LIN {X 0,Y 227.48,Z 413.452,A -85,B 0,C 180,E1 -20071.549,E2 -20071.549} C_VEL
LIN {X 0,Y 229.431,Z 419.011,A -85,B 0,C 180,E1 -20072.113,E2 -20072.113} C_VEL
LIN {X 0,Y 232.669,Z 428.465,A -85,B 0,C 180,E1 -20073.214,E2 -20073.214} C_VEL
LIN {X 0,Y 235.611,Z 440.17,A -85,B 0,C 180,E1 -20074.705,E2 -20074.705} C_VEL
LIN {X 0,Y 237.998,Z 451.953,A -85,B 0,C 180,E1 -20076.482,E2 -20076.482} C_VEL
LIN {X 0,Y 238.523,Z 456.323,A -85,B 0,C 180,E1 -20077.194,E2 -20077.194} C_VEL
LIN {X 0,Y 236.555,Z 467.31,A -85,B 0,C 180,E1 -20078.946,E2 -20078.946} C_VEL
LIN {X 0,Y 234.438,Z 477.678,A -85,B 0,C 180,E1 -20081.018,E2 -20081.018} C_VEL
LIN {X 0,Y 232.639,Z 485.999,A -85,B 0,C 180,E1 -20083.096,E2 -20083.096} C_VEL
LIN {X 0,Y 230.834,Z 493.681,A -85,B 0,C 180,E1 -20085.45,E2 -20085.45} C_VEL
LIN {X 0,Y 229.18,Z 500.557,A -85,B 0,C 180,E1 -20088.076,E2 -20088.076} C_VEL
LIN {X 0,Y 227.975,Z 506.106,A -85,B 0,C 180,E1 -20090.764,E2 -20090.764} C_VEL
LIN {X 0,Y 226.971,Z 510.814,A -85,B 0,C 180,E1 -20093.737,E2 -20093.737} C_VEL
LIN {X 0,Y 226.477,Z 513.304,A -85,B 0,C 180,E1 -20095.851,E2 -20095.851} C_VEL
LIN {X 0,Y 226.081,Z 515.094,A -85,B 0,C 180,E1 -20097.794,E2 -20097.794} C_VEL
LIN {X 0,Y 225.853,Z 516.41,A -85,B 0,C 180,E1 -20099.86,E2 -20099.86} C_VEL
LIN {X 0,Y 225.805,Z 517.379,A -85,B 0,C 180,E1 -20102.822,E2 -20102.822} C_VEL
LIN {X 0,Y 226.172,Z 517.171,A -85,B 0,C 180,E1 -20106.185,E2 -20106.185} C_VEL
LIN {X 0,Y 226.927,Z 515.743,A -85,B 0,C 180,E1 -20109.262,E2 -20109.262} C_VEL
LIN {X 0,Y 228.213,Z 512.694,A -85,B 0,C 180,E1 -20112.649,E2 -20112.649} C_VEL
LIN {X 0,Y 229.437,Z 509.335,A -85,B 0,C 180,E1 -20115.208,E2 -20115.208} C_VEL
LIN {X 0,Y 231.319,Z 504.308,A -85,B 0,C 180,E1 -20118.055,E2 -20118.055} C_VEL
LIN {X 0,Y 233.64,Z 497.907,A -85,B 0,C 180,E1 -20120.825,E2 -20120.825} C_VEL
LIN {X 0,Y 236.35,Z 489.874,A -85,B 0,C 180,E1 -20123.508,E2 -20123.508} C_VEL
LIN {X 0,Y 239.203,Z 480.611,A -85,B 0,C 180,E1 -20125.926,E2 -20125.926} C_VEL
LIN {X 0,Y 241.778,Z 471.395,A -85,B 0,C 180,E1 -20127.84,E2 -20127.84} C_VEL
LIN {X 0,Y 243.706,Z 463.116,A -85,B 0,C 180,E1 -20129.259,E2 -20129.259} C_VEL
LIN {X 0,Y 242.372,Z 453.565,A -85,B 0,C 180,E1 -20131.179,E2 -20131.179} C_VEL
LIN {X 0,Y 240.028,Z 444.017,A -85,B 0,C 180,E1 -20133.009,E2 -20133.009} C_VEL
LIN {X 0,Y 237.284,Z 435.697,A -85,B 0,C 180,E1 -20134.566,E2 -20134.566} C_VEL
LIN {X 0,Y 232.657,Z 425.144,A -85,B 0,C 180,E1 -20136.583,E2 -20136.583} C_VEL
LIN {X 0,Y 230.235,Z 420.752,A -85,B 0,C 180,E1 -20137.483,E2 -20137.483} C_VEL
LIN {X 0,Y 228.674,Z 417.665,A -85,B 0,C 180,E1 -20138.078,E2 -20138.078} C_VEL
LIN {X 0,Y 228.509,Z 416.855,A -85,B 0,C 180,E1 -20138.248,E2 -20138.248} C_VEL
LIN {X 0,Y 228.454,Z 415.047,A -85,B 0,C 180,E1 -20142.487,E2 -20142.487} C_VEL
LIN {X 0,Y 228.344,Z 413.795,A -85,B 0,C 180,E1 -20145.745,E2 -20145.745} C_VEL
LIN {X 0,Y 228.264,Z 412.058,A -85,B 0,C 180,E1 -20151.144,E2 -20151.144} C_VEL
LIN {X 0,Y 228.322,Z 412.042,A -85,B 0,C 180,E1 -20152.927,E2 -20152.927} C_VEL
LIN {X 0,Y 228.552,Z 412.016,A -85,B 0,C 180,E1 -20158.238,E2 -20158.238} C_VEL
LIN {X 0,Y 228.552,Z 412.013,A -85,B 0,C 180,E1 -20161.762,E2 -20161.762} C_VEL
LIN {X 0,Y 228.321,Z 412.042,A -85,B 0,C 180,E1 -20167.072,E2 -20167.072} C_VEL
LIN {X 0,Y 228.143,Z 412.061,A -85,B 0,C 180,E1 -20170.651,E2 -20170.651} C_VEL
LIN {X 0,Y 228.06,Z 412.073,A -85,B 0,C 180,E1 -20174.272,E2 -20174.272} C_VEL
LIN {X 0,Y 228.001,Z 412.082,A -85,B 0,C 180,E1 -20177.953,E2 -20177.953} C_VEL
LIN {X 0,Y 227.994,Z 412.377,A -85,B 0,C 180,E1 -20182.369,E2 -20182.369} C_VEL
LIN {X 0,Y 228.285,Z 414.087,A -85,B 0,C 180,E1 -20186.775,E2 -20186.775} C_VEL
LIN {X 0,Y 228.651,Z 416.429,A -85,B 0,C 180,E1 -20191.502,E2 -20191.502} C_VEL
LIN {X 0,Y 228.94,Z 417.889,A -85,B 0,C 180,E1 -20194.02,E2 -20194.02} C_VEL
LIN {X 0,Y 229.338,Z 420.345,A -85,B 0,C 180,E1 -20197.799,E2 -20197.799} C_VEL
LIN {X 0,Y 229.909,Z 423.677,A -85,B 0,C 180,E1 -20202.261,E2 -20202.261} C_VEL
LIN {X 0,Y 230.662,Z 427.668,A -85,B 0,C 180,E1 -20206.991,E2 -20206.991} C_VEL
LIN {X 0,Y 231.147,Z 430.792,A -85,B 0,C 180,E1 -20210.32,E2 -20210.32} C_VEL
LIN {X 0,Y 231.208,Z 433.067,A -85,B 0,C 180,E1 -20212.56,E2 -20212.56} C_VEL
LIN {X 0,Y 230.752,Z 434.935,A -85,B 0,C 180,E1 -20214.276,E2 -20214.276} C_VEL
LIN {X 0,Y 231.711,Z 438.454,A -85,B 0,C 180,E1 -20214.705,E2 -20214.705} C_VEL
LIN {X 0,Y 232.658,Z 441.188,A -85,B 0,C 180,E1 -20215.093,E2 -20215.093} C_VEL
LIN {X 0,Y 235.69,Z 451.302,A -85,B 0,C 180,E1 -20216.544,E2 -20216.544} C_VEL
LIN {X 0,Y 236.026,Z 456.772,A -85,B 0,C 180,E1 -20217.157,E2 -20217.157} C_VEL
LIN {X 0,Y 234.94,Z 466.073,A -85,B 0,C 180,E1 -20218.079,E2 -20218.079} C_VEL
LIN {X 0,Y 233.754,Z 473.124,A -85,B 0,C 180,E1 -20218.886,E2 -20218.886} C_VEL
LIN {X 0,Y 233.258,Z 479.739,A -85,B 0,C 180,E1 -20219.88,E2 -20219.88} C_VEL
LIN {X 0,Y 232.962,Z 490.074,A -85,B 0,C 180,E1 -20221.784,E2 -20221.784} C_VEL
LIN {X 0,Y 231.795,Z 500.22,A -85,B 0,C 180,E1 -20223.919,E2 -20223.919} C_VEL
LIN {X 0,Y 229.01,Z 509.22,A -85,B 0,C 180,E1 -20226.007,E2 -20226.007} C_VEL
LIN {X 0,Y 226.204,Z 517.822,A -85,B 0,C 180,E1 -20228.499,E2 -20228.499} C_VEL
LIN {X 0,Y 223.821,Z 525.268,A -85,B 0,C 180,E1 -20231.225,E2 -20231.225} C_VEL
LIN {X 0,Y 221.61,Z 531.902,A -85,B 0,C 180,E1 -20234.362,E2 -20234.362} C_VEL
LIN {X 0,Y 220.174,Z 536.342,A -85,B 0,C 180,E1 -20237.089,E2 -20237.089} C_VEL
LIN {X 0,Y 219.588,Z 538.722,A -85,B 0,C 180,E1 -20238.928,E2 -20238.928} C_VEL
LIN {X 0,Y 219.114,Z 540.678,A -85,B 0,C 180,E1 -20240.771,E2 -20240.771} C_VEL
LIN {X 0,Y 218.857,Z 542.179,A -85,B 0,C 180,E1 -20242.62,E2 -20242.62} C_VEL
LIN {X 0,Y 218.739,Z 543.478,A -85,B 0,C 180,E1 -20244.885,E2 -20244.885} C_VEL
LIN {X 0,Y 218.819,Z 544.309,A -85,B 0,C 180,E1 -20248.159,E2 -20248.159} C_VEL
LIN {X 0,Y 218.888,Z 544.196,A -85,B 0,C 180,E1 -20250,E2 -20250} C_VEL
LIN {X 0,Y 218.843,Z 543.657,A -85,B 0,C 180,E1 -20251.84,E2 -20251.84} C_VEL
LIN {X 0,Y 218.813,Z 542.715,A -85,B 0,C 180,E1 -20253.683,E2 -20253.683} C_VEL
LIN {X 0,Y 218.886,Z 541.368,A -85,B 0,C 180,E1 -20255.527,E2 -20255.527} C_VEL
LIN {X 0,Y 219.041,Z 538.468,A -85,B 0,C 180,E1 -20258.301,E2 -20258.301} C_VEL
LIN {X 0,Y 219.603,Z 534.518,A -85,B 0,C 180,E1 -20261.07,E2 -20261.07} C_VEL
LIN {X 0,Y 220.721,Z 528.412,A -85,B 0,C 180,E1 -20264.286,E2 -20264.286} C_VEL
LIN {X 0,Y 222.266,Z 521.731,A -85,B 0,C 180,E1 -20267.006,E2 -20267.006} C_VEL
LIN {X 0,Y 223.85,Z 515.198,A -85,B 0,C 180,E1 -20269.162,E2 -20269.162} C_VEL
LIN {X 0,Y 225.679,Z 506.899,A -85,B 0,C 180,E1 -20271.415,E2 -20271.415} C_VEL
LIN {X 0,Y 227.98,Z 496.745,A -85,B 0,C 180,E1 -20273.624,E2 -20273.624} C_VEL
LIN {X 0,Y 228.308,Z 489.287,A -85,B 0,C 180,E1 -20275.04,E2 -20275.04} C_VEL
LIN {X 0,Y 227.969,Z 478.102,A -85,B 0,C 180,E1 -20276.898,E2 -20276.898} C_VEL
LIN {X 0,Y 226.994,Z 466.517,A -85,B 0,C 180,E1 -20278.508,E2 -20278.508} C_VEL
LIN {X 0,Y 225.199,Z 453.339,A -85,B 0,C 180,E1 -20280.012,E2 -20280.012} C_VEL
LIN {X 0,Y 222.537,Z 439.898,A -85,B 0,C 180,E1 -20281.269,E2 -20281.269} C_VEL
LIN {X 0,Y 222.063,Z 437.235,A -85,B 0,C 180,E1 -20281.501,E2 -20281.501} C_VEL
LIN {X 0,Y 223.062,Z 433.147,A -85,B 0,C 180,E1 -20284.997,E2 -20284.997} C_VEL
LIN {X 0,Y 223.543,Z 431.209,A -85,B 0,C 180,E1 -20286.678,E2 -20286.678} C_VEL
LIN {X 0,Y 223.678,Z 428.7,A -85,B 0,C 180,E1 -20288.931,E2 -20288.931} C_VEL
LIN {X 0,Y 223.07,Z 425.028,A -85,B 0,C 180,E1 -20292.459,E2 -20292.459} C_VEL
LIN {X 0,Y 222.261,Z 420.887,A -85,B 0,C 180,E1 -20296.656,E2 -20296.656} C_VEL
LIN {X 0,Y 221.568,Z 417.22,A -85,B 0,C 180,E1 -20300.625,E2 -20300.625} C_VEL
LIN {X 0,Y 220.972,Z 413.335,A -85,B 0,C 180,E1 -20305.076,E2 -20305.076} C_VEL
LIN {X 0,Y 220.867,Z 412.973,A -85,B 0,C 180,E1 -20305.822,E2 -20305.822} C_VEL
LIN {X 0,Y 220.864,Z 412.976,A -85,B 0,C 180,E1 -20309.394,E2 -20309.394} C_VEL
LIN {X 0,Y 220.891,Z 412.97,A -85,B 0,C 180,E1 -20313.549,E2 -20313.549} C_VEL
LIN {X 0,Y 220.873,Z 412.971,A -85,B 0,C 180,E1 -20317.553,E2 -20317.553} C_VEL
LIN {X 0,Y 220.979,Z 412.96,A -85,B 0,C 180,E1 -20322.571,E2 -20322.571} C_VEL
LIN {X 0,Y 221.006,Z 412.955,A -85,B 0,C 180,E1 -20327.138,E2 -20327.138} C_VEL
LIN {X 0,Y 221.199,Z 412.931,A -85,B 0,C 180,E1 -20330.859,E2 -20330.859} C_VEL
LIN {X 0,Y 221.253,Z 412.92,A -85,B 0,C 180,E1 -20332.701,E2 -20332.701} C_VEL
LIN {X 0,Y 221.507,Z 412.892,A -85,B 0,C 180,E1 -20338.182,E2 -20338.182} C_VEL
LIN {X 0,Y 221.507,Z 412.887,A -85,B 0,C 180,E1 -20341.818,E2 -20341.818} C_VEL
LIN {X 0,Y 221.284,Z 412.919,A -85,B 0,C 180,E1 -20347.299,E2 -20347.299} C_VEL
LIN {X 0,Y 221.107,Z 412.937,A -85,B 0,C 180,E1 -20350.995,E2 -20350.995} C_VEL
LIN {X 0,Y 221.011,Z 412.956,A -85,B 0,C 180,E1 -20356.63,E2 -20356.63} C_VEL
LIN {X 0,Y 220.888,Z 412.967,A -85,B 0,C 180,E1 -20360.487,E2 -20360.487} C_VEL
LIN {X 0,Y 220.863,Z 412.967,A -85,B 0,C 180,E1 -20364.436,E2 -20364.436} C_VEL
LIN {X 0,Y 220.833,Z 412.977,A -85,B 0,C 180,E1 -20368.514,E2 -20368.514} C_VEL
LIN {X 0,Y 220.821,Z 412.971,A -85,B 0,C 180,E1 -20372.756,E2 -20372.756} C_VEL
LIN {X 0,Y 220.836,Z 412.975,A -85,B 0,C 180,E1 -20377.289,E2 -20377.289} C_VEL
LIN {X 0,Y 220.785,Z 412.975,A -85,B 0,C 180,E1 -20381.95,E2 -20381.95} C_VEL
LIN {X 0,Y 220.773,Z 412.984,A -85,B 0,C 180,E1 -20385.547,E2 -20385.547} C_VEL
LIN {X 0,Y 220.805,Z 412.963,A -85,B 0,C 180,E1 -20390.464,E2 -20390.464} C_VEL
LIN {X 0,Y 220.8,Z 412.973,A -85,B 0,C 180,E1 -20395.046,E2 -20395.046} C_VEL
LIN {X 0,Y 220.834,Z 412.979,A -85,B 0,C 180,E1 -20399.391,E2 -20399.391} C_VEL
LIN {X 0,Y 220.895,Z 412.957,A -85,B 0,C 180,E1 -20403.551,E2 -20403.551} C_VEL
LIN {X 0,Y 220.879,Z 412.969,A -85,B 0,C 180,E1 -20407.555,E2 -20407.555} C_VEL
LIN {X 0,Y 220.986,Z 412.946,A -85,B 0,C 180,E1 -20412.572,E2 -20412.572} C_VEL
LIN {X 0,Y 221.029,Z 412.953,A -85,B 0,C 180,E1 -20417.14,E2 -20417.14} C_VEL
LIN {X 0,Y 221.261,Z 412.923,A -85,B 0,C 180,E1 -20420.862,E2 -20420.862} C_VEL
LIN {X 0,Y 221.312,Z 412.917,A -85,B 0,C 180,E1 -20422.703,E2 -20422.703} C_VEL
LIN {X 0,Y 221.332,Z 412.916,A -85,B 0,C 180,E1 -20428.181,E2 -20428.181} C_VEL
LIN {X 0,Y 220.566,Z 413.818,A -85,B 0,C 180,E1 -20430.628,E2 -20430.628} C_VEL
LIN {X 0,Y 222.442,Z 419.58,A -85,B 0,C 180,E1 -20431.273,E2 -20431.273} C_VEL
LIN {X 0,Y 226.158,Z 430.27,A -85,B 0,C 180,E1 -20432.583,E2 -20432.583} C_VEL
LIN {X 0,Y 228.879,Z 440.962,A -85,B 0,C 180,E1 -20434.031,E2 -20434.031} C_VEL
LIN {X 0,Y 231.193,Z 452.796,A -85,B 0,C 180,E1 -20435.889,E2 -20435.889} C_VEL
LIN {X 0,Y 231.741,Z 457.845,A -85,B 0,C 180,E1 -20436.749,E2 -20436.749} C_VEL
LIN {X 0,Y 229.642,Z 468.84,A -85,B 0,C 180,E1 -20438.581,E2 -20438.581} C_VEL
LIN {X 0,Y 227.495,Z 478.832,A -85,B 0,C 180,E1 -20440.682,E2 -20440.682} C_VEL
LIN {X 0,Y 225.422,Z 487.746,A -85,B 0,C 180,E1 -20443.027,E2 -20443.027} C_VEL
LIN {X 0,Y 223.627,Z 495.303,A -85,B 0,C 180,E1 -20445.494,E2 -20445.494} C_VEL
LIN {X 0,Y 221.899,Z 502.52,A -85,B 0,C 180,E1 -20448.465,E2 -20448.465} C_VEL
LIN {X 0,Y 220.599,Z 507.98,A -85,B 0,C 180,E1 -20451.392,E2 -20451.392} C_VEL
LIN {X 0,Y 219.703,Z 512.413,A -85,B 0,C 180,E1 -20454.573,E2 -20454.573} C_VEL
LIN {X 0,Y 219.204,Z 514.599,A -85,B 0,C 180,E1 -20456.671,E2 -20456.671} C_VEL
LIN {X 0,Y 218.764,Z 516.808,A -85,B 0,C 180,E1 -20459.841,E2 -20459.841} C_VEL
LIN {X 0,Y 218.75,Z 517.869,A -85,B 0,C 180,E1 -20463.349,E2 -20463.349} C_VEL
LIN {X 0,Y 219.198,Z 517.556,A -85,B 0,C 180,E1 -20466.72,E2 -20466.72} C_VEL
LIN {X 0,Y 220.052,Z 515.969,A -85,B 0,C 180,E1 -20469.958,E2 -20469.958} C_VEL
LIN {X 0,Y 221.287,Z 513.217,A -85,B 0,C 180,E1 -20473.073,E2 -20473.073} C_VEL
LIN {X 0,Y 223.055,Z 508.776,A -85,B 0,C 180,E1 -20476.442,E2 -20476.442} C_VEL
LIN {X 0,Y 224.945,Z 504.166,A -85,B 0,C 180,E1 -20478.996,E2 -20478.996} C_VEL
LIN {X 0,Y 227.367,Z 497.674,A -85,B 0,C 180,E1 -20481.814,E2 -20481.814} C_VEL
LIN {X 0,Y 230.326,Z 489.39,A -85,B 0,C 180,E1 -20484.566,E2 -20484.566} C_VEL
LIN {X 0,Y 232.963,Z 481.172,A -85,B 0,C 180,E1 -20486.748,E2 -20486.748} C_VEL
LIN {X 0,Y 235.967,Z 470.937,A -85,B 0,C 180,E1 -20488.901,E2 -20488.901} C_VEL
LIN {X 0,Y 237.27,Z 466.006,A -85,B 0,C 180,E1 -20489.765,E2 -20489.765} C_VEL
LIN {X 0,Y 237.023,Z 460.903,A -85,B 0,C 180,E1 -20490.83,E2 -20490.83} C_VEL
LIN {X 0,Y 235.16,Z 450.402,A -85,B 0,C 180,E1 -20493.006,E2 -20493.006} C_VEL
LIN {X 0,Y 232.04,Z 439.785,A -85,B 0,C 180,E1 -20495.165,E2 -20495.165} C_VEL
LIN {X 0,Y 227.861,Z 429.694,A -85,B 0,C 180,E1 -20497.253,E2 -20497.253} C_VEL
LIN {X 0,Y 223.672,Z 421.792,A -85,B 0,C 180,E1 -20498.998,E2 -20498.998} C_VEL
LIN {X 0,Y 221.912,Z 418.938,A -85,B 0,C 180,E1 -20499.672,E2 -20499.672} C_VEL
LIN {X 0,Y 221.522,Z 417.488,A -85,B 0,C 180,E1 -20499.938,E2 -20499.938} C_VEL
LIN {X 0,Y 221.453,Z 416.115,A -85,B 0,C 180,E1 -20503.404,E2 -20503.404} C_VEL
LIN {X 0,Y 221.326,Z 414.816,A -85,B 0,C 180,E1 -20507.157,E2 -20507.157} C_VEL
LIN {X 0,Y 221.328,Z 413.693,A -85,B 0,C 180,E1 -20510.864,E2 -20510.864} C_VEL
LIN {X 0,Y 221.299,Z 413.218,A -85,B 0,C 180,E1 -20512.702,E2 -20512.702} C_VEL
LIN {X 0,Y 221.51,Z 412.892,A -85,B 0,C 180,E1 -20518.182,E2 -20518.182} C_VEL
LIN {X 0,Y 221.51,Z 412.889,A -85,B 0,C 180,E1 -20521.818,E2 -20521.818} C_VEL
LIN {X 0,Y 221.257,Z 412.92,A -85,B 0,C 180,E1 -20527.299,E2 -20527.299} C_VEL
LIN {X 0,Y 221.065,Z 412.942,A -85,B 0,C 180,E1 -20530.996,E2 -20530.996} C_VEL
LIN {X 0,Y 221.014,Z 412.949,A -85,B 0,C 180,E1 -20536.63,E2 -20536.63} C_VEL
LIN {X 0,Y 220.92,Z 413.037,A -85,B 0,C 180,E1 -20538.549,E2 -20538.549} C_VEL
LIN {X 0,Y 221.138,Z 414.298,A -85,B 0,C 180,E1 -20542.833,E2 -20542.833} C_VEL
LIN {X 0,Y 221.427,Z 416.044,A -85,B 0,C 180,E1 -20547.29,E2 -20547.29} C_VEL
LIN {X 0,Y 221.74,Z 417.919,A -85,B 0,C 180,E1 -20551.158,E2 -20551.158} C_VEL
LIN {X 0,Y 222.1,Z 419.925,A -85,B 0,C 180,E1 -20554.721,E2 -20554.721} C_VEL
LIN {X 0,Y 222.541,Z 422.862,A -85,B 0,C 180,E1 -20559.169,E2 -20559.169} C_VEL
LIN {X 0,Y 223.161,Z 426.398,A -85,B 0,C 180,E1 -20563.856,E2 -20563.856} C_VEL
LIN {X 0,Y 223.762,Z 429.514,A -85,B 0,C 180,E1 -20567.555,E2 -20567.555} C_VEL
LIN {X 0,Y 224.154,Z 431.757,A -85,B 0,C 180,E1 -20570.042,E2 -20570.042} C_VEL
LIN {X 0,Y 224.16,Z 434.343,A -85,B 0,C 180,E1 -20572.671,E2 -20572.671} C_VEL
LIN {X 0,Y 225.061,Z 437.718,A -85,B 0,C 180,E1 -20573.138,E2 -20573.138} C_VEL
LIN {X 0,Y 225.989,Z 439.903,A -85,B 0,C 180,E1 -20573.518,E2 -20573.518} C_VEL
LIN {X 0,Y 229.36,Z 451.137,A -85,B 0,C 180,E1 -20575.256,E2 -20575.256} C_VEL
LIN {X 0,Y 231.934,Z 463.884,A -85,B 0,C 180,E1 -20577.233,E2 -20577.233} C_VEL
LIN {X 0,Y 233.077,Z 475.66,A -85,B 0,C 180,E1 -20579.163,E2 -20579.163} C_VEL
LIN {X 0,Y 233.258,Z 479.739,A -85,B 0,C 180,E1 -20579.88,E2 -20579.88} C_VEL
LIN {X 0,Y 232.713,Z 484.647,A -85,B 0,C 180,E1 -20580.674,E2 -20580.674} C_VEL
LIN {X 0,Y 231.139,Z 489.559,A -85,B 0,C 180,E1 -20581.407,E2 -20581.407} C_VEL
LIN {X 0,Y 226.67,Z 499.013,A -85,B 0,C 180,E1 -20582.91,E2 -20582.91} C_VEL
LIN {X 0,Y 224.134,Z 504.879,A -85,B 0,C 180,E1 -20584.134,E2 -20584.134} C_VEL
LIN {X 0,Y 220.951,Z 513.992,A -85,B 0,C 180,E1 -20586.572,E2 -20586.572} C_VEL
LIN {X 0,Y 218.32,Z 521.861,A -85,B 0,C 180,E1 -20589.261,E2 -20589.261} C_VEL
LIN {X 0,Y 216.029,Z 528.216,A -85,B 0,C 180,E1 -20591.997,E2 -20591.997} C_VEL
LIN {X 0,Y 214.163,Z 533.328,A -85,B 0,C 180,E1 -20594.78,E2 -20594.78} C_VEL
LIN {X 0,Y 212.878,Z 537.346,A -85,B 0,C 180,E1 -20597.608,E2 -20597.608} C_VEL
LIN {X 0,Y 212.081,Z 540.369,A -85,B 0,C 180,E1 -20600.462,E2 -20600.462} C_VEL
LIN {X 0,Y 211.657,Z 542.905,A -85,B 0,C 180,E1 -20604.283,E2 -20604.283} C_VEL
LIN {X 0,Y 211.645,Z 543.59,A -85,B 0,C 180,E1 -20606.192,E2 -20606.192} C_VEL
LIN {X 0,Y 211.749,Z 543.878,A -85,B 0,C 180,E1 -20608.098,E2 -20608.098} C_VEL
LIN {X 0,Y 211.817,Z 543.722,A -85,B 0,C 180,E1 -20610,E2 -20610} C_VEL
LIN {X 0,Y 211.775,Z 543.156,A -85,B 0,C 180,E1 -20611.901,E2 -20611.901} C_VEL
LIN {X 0,Y 211.788,Z 541.031,A -85,B 0,C 180,E1 -20615.424,E2 -20615.424} C_VEL
LIN {X 0,Y 212,Z 537.852,A -85,B 0,C 180,E1 -20618.579,E2 -20618.579} C_VEL
LIN {X 0,Y 212.595,Z 533.839,A -85,B 0,C 180,E1 -20621.44,E2 -20621.44} C_VEL
LIN {X 0,Y 213.819,Z 527.637,A -85,B 0,C 180,E1 -20624.757,E2 -20624.757} C_VEL
LIN {X 0,Y 215.435,Z 520.877,A -85,B 0,C 180,E1 -20627.562,E2 -20627.562} C_VEL
LIN {X 0,Y 216.987,Z 514.628,A -85,B 0,C 180,E1 -20629.669,E2 -20629.669} C_VEL
LIN {X 0,Y 219.059,Z 505.677,A -85,B 0,C 180,E1 -20632.145,E2 -20632.145} C_VEL
LIN {X 0,Y 221.342,Z 495.518,A -85,B 0,C 180,E1 -20634.378,E2 -20634.378} C_VEL
LIN {X 0,Y 221.353,Z 485.038,A -85,B 0,C 180,E1 -20636.39,E2 -20636.39} C_VEL
LIN {X 0,Y 220.825,Z 473.117,A -85,B 0,C 180,E1 -20638.304,E2 -20638.304} C_VEL
LIN {X 0,Y 219.496,Z 460.966,A -85,B 0,C 180,E1 -20639.945,E2 -20639.945} C_VEL
LIN {X 0,Y 217.597,Z 448.69,A -85,B 0,C 180,E1 -20641.299,E2 -20641.299} C_VEL
LIN {X 0,Y 215.195,Z 436.842,A -85,B 0,C 180,E1 -20642.411,E2 -20642.411} C_VEL
LIN {X 0,Y 216.523,Z 431.771,A -85,B 0,C 180,E1 -20646.903,E2 -20646.903} C_VEL
LIN {X 0,Y 216.64,Z 429.657,A -85,B 0,C 180,E1 -20648.869,E2 -20648.869} C_VEL
LIN {X 0,Y 215.908,Z 425.361,A -85,B 0,C 180,E1 -20653.121,E2 -20653.121} C_VEL
LIN {X 0,Y 215.247,Z 421.951,A -85,B 0,C 180,E1 -20656.712,E2 -20656.712} C_VEL
LIN {X 0,Y 214.384,Z 417.36,A -85,B 0,C 180,E1 -20661.883,E2 -20661.883} C_VEL
LIN {X 0,Y 213.802,Z 413.854,A -85,B 0,C 180,E1 -20666.168,E2 -20666.168} C_VEL
LIN {X 0,Y 213.776,Z 413.859,A -85,B 0,C 180,E1 -20670.453,E2 -20670.453} C_VEL
LIN {X 0,Y 213.797,Z 413.856,A -85,B 0,C 180,E1 -20674.701,E2 -20674.701} C_VEL
LIN {X 0,Y 213.808,Z 413.854,A -85,B 0,C 180,E1 -20678.803,E2 -20678.803} C_VEL
LIN {X 0,Y 213.939,Z 413.837,A -85,B 0,C 180,E1 -20682.803,E2 -20682.803} C_VEL
LIN {X 0,Y 213.948,Z 413.836,A -85,B 0,C 180,E1 -20686.706,E2 -20686.706} C_VEL
LIN {X 0,Y 214.137,Z 413.812,A -85,B 0,C 180,E1 -20690.555,E2 -20690.555} C_VEL
LIN {X 0,Y 214.095,Z 413.808,A -85,B 0,C 180,E1 -20694.349,E2 -20694.349} C_VEL
LIN {X 0,Y 214.44,Z 413.772,A -85,B 0,C 180,E1 -20698.122,E2 -20698.122} C_VEL
LIN {X 0,Y 214.549,Z 413.758,A -85,B 0,C 180,E1 -20700,E2 -20700} C_VEL
LIN {X 0,Y 214.44,Z 413.768,A -85,B 0,C 180,E1 -20701.878,E2 -20701.878} C_VEL
LIN {X 0,Y 214.222,Z 413.799,A -85,B 0,C 180,E1 -20707.541,E2 -20707.541} C_VEL
LIN {X 0,Y 214.039,Z 413.816,A -85,B 0,C 180,E1 -20711.362,E2 -20711.362} C_VEL
LIN {X 0,Y 213.927,Z 413.833,A -85,B 0,C 180,E1 -20715.238,E2 -20715.238} C_VEL
LIN {X 0,Y 213.835,Z 413.846,A -85,B 0,C 180,E1 -20719.188,E2 -20719.188} C_VEL
LIN {X 0,Y 213.843,Z 413.836,A -85,B 0,C 180,E1 -20723.228,E2 -20723.228} C_VEL
LIN {X 0,Y 213.826,Z 413.848,A -85,B 0,C 180,E1 -20727.451,E2 -20727.451} C_VEL
LIN {X 0,Y 213.776,Z 413.849,A -85,B 0,C 180,E1 -20731.737,E2 -20731.737} C_VEL
LIN {X 0,Y 213.751,Z 413.86,A -85,B 0,C 180,E1 -20736.287,E2 -20736.287} C_VEL
LIN {X 0,Y 213.722,Z 413.852,A -85,B 0,C 180,E1 -20741.123,E2 -20741.123} C_VEL
LIN {X 0,Y 213.728,Z 413.86,A -85,B 0,C 180,E1 -20743.673,E2 -20743.673} C_VEL
LIN {X 0,Y 213.705,Z 413.865,A -85,B 0,C 180,E1 -20746.345,E2 -20746.345} C_VEL
LIN {X 0,Y 213.716,Z 413.854,A -85,B 0,C 180,E1 -20749.144,E2 -20749.144} C_VEL
LIN {X 0,Y 213.743,Z 413.839,A -85,B 0,C 180,E1 -20753.713,E2 -20753.713} C_VEL
LIN {X 0,Y 213.78,Z 413.858,A -85,B 0,C 180,E1 -20758.733,E2 -20758.733} C_VEL
LIN {X 0,Y 213.827,Z 413.841,A -85,B 0,C 180,E1 -20762.604,E2 -20762.604} C_VEL
LIN {X 0,Y 213.853,Z 413.842,A -85,B 0,C 180,E1 -20766.954,E2 -20766.954} C_VEL
LIN {X 0,Y 213.946,Z 413.822,A -85,B 0,C 180,E1 -20772.805,E2 -20772.805} C_VEL
LIN {X 0,Y 213.983,Z 413.83,A -85,B 0,C 180,E1 -20776.709,E2 -20776.709} C_VEL
LIN {X 0,Y 214.2,Z 413.804,A -85,B 0,C 180,E1 -20780.558,E2 -20780.558} C_VEL
LIN {X 0,Y 214.249,Z 413.797,A -85,B 0,C 180,E1 -20782.461,E2 -20782.461} C_VEL
LIN {X 0,Y 214.283,Z 413.794,A -85,B 0,C 180,E1 -20788.121,E2 -20788.121} C_VEL
LIN {X 0,Y 213.693,Z 414.194,A -85,B 0,C 180,E1 -20789.647,E2 -20789.647} C_VEL
LIN {X 0,Y 213.686,Z 414.29,A -85,B 0,C 180,E1 -20789.765,E2 -20789.765} C_VEL
LIN {X 0,Y 216.06,Z 421.684,A -85,B 0,C 180,E1 -20790.577,E2 -20790.577} C_VEL
LIN {X 0,Y 219.971,Z 433.168,A -85,B 0,C 180,E1 -20792.099,E2 -20792.099} C_VEL
LIN {X 0,Y 222.537,Z 443.678,A -85,B 0,C 180,E1 -20793.622,E2 -20793.622} C_VEL
LIN {X 0,Y 224.759,Z 455.6,A -85,B 0,C 180,E1 -20795.608,E2 -20795.608} C_VEL
LIN {X 0,Y 225.068,Z 457.987,A -85,B 0,C 180,E1 -20796.05,E2 -20796.05} C_VEL
LIN {X 0,Y 223.033,Z 468.93,A -85,B 0,C 180,E1 -20797.924,E2 -20797.924} C_VEL
LIN {X 0,Y 220.959,Z 478.381,A -85,B 0,C 180,E1 -20799.934,E2 -20799.934} C_VEL
LIN {X 0,Y 219.064,Z 486.422,A -85,B 0,C 180,E1 -20802.037,E2 -20802.037} C_VEL
LIN {X 0,Y 217.131,Z 494.051,A -85,B 0,C 180,E1 -20804.48,E2 -20804.48} C_VEL
LIN {X 0,Y 215.471,Z 500.583,A -85,B 0,C 180,E1 -20807.071,E2 -20807.071} C_VEL
LIN {X 0,Y 213.984,Z 506.733,A -85,B 0,C 180,E1 -20810.173,E2 -20810.173} C_VEL
LIN {X 0,Y 212.893,Z 511.496,A -85,B 0,C 180,E1 -20813.337,E2 -20813.337} C_VEL
LIN {X 0,Y 212.128,Z 514.962,A -85,B 0,C 180,E1 -20816.55,E2 -20816.55} C_VEL
LIN {X 0,Y 211.667,Z 517.425,A -85,B 0,C 180,E1 -20820.312,E2 -20820.312} C_VEL
LIN {X 0,Y 211.702,Z 518.357,A -85,B 0,C 180,E1 -20823.906,E2 -20823.906} C_VEL
LIN {X 0,Y 212.228,Z 517.894,A -85,B 0,C 180,E1 -20827.366,E2 -20827.366} C_VEL
LIN {X 0,Y 213.2,Z 516.192,A -85,B 0,C 180,E1 -20830.695,E2 -20830.695} C_VEL
LIN {X 0,Y 214.563,Z 513.345,A -85,B 0,C 180,E1 -20833.895,E2 -20833.895} C_VEL
LIN {X 0,Y 216.246,Z 509.383,A -85,B 0,C 180,E1 -20836.96,E2 -20836.96} C_VEL
LIN {X 0,Y 218.544,Z 504.095,A -85,B 0,C 180,E1 -20839.971,E2 -20839.971} C_VEL
LIN {X 0,Y 221.238,Z 497.374,A -85,B 0,C 180,E1 -20842.874,E2 -20842.874} C_VEL
LIN {X 0,Y 224.369,Z 488.986,A -85,B 0,C 180,E1 -20845.679,E2 -20845.679} C_VEL
LIN {X 0,Y 227.316,Z 480.188,A -85,B 0,C 180,E1 -20847.996,E2 -20847.996} C_VEL
LIN {X 0,Y 230.212,Z 470.563,A -85,B 0,C 180,E1 -20849.998,E2 -20849.998} C_VEL
LIN {X 0,Y 231.11,Z 467.205,A -85,B 0,C 180,E1 -20850.612,E2 -20850.612} C_VEL
LIN {X 0,Y 230.423,Z 459.571,A -85,B 0,C 180,E1 -20852.33,E2 -20852.33} C_VEL
LIN {X 0,Y 228.922,Z 451.733,A -85,B 0,C 180,E1 -20854.056,E2 -20854.056} C_VEL
LIN {X 0,Y 226.118,Z 442.018,A -85,B 0,C 180,E1 -20856.168,E2 -20856.168} C_VEL
LIN {X 0,Y 222.444,Z 433.051,A -85,B 0,C 180,E1 -20858.208,E2 -20858.208} C_VEL
LIN {X 0,Y 219.117,Z 426.506,A -85,B 0,C 180,E1 -20859.769,E2 -20859.769} C_VEL
LIN {X 0,Y 216.983,Z 422.612,A -85,B 0,C 180,E1 -20860.733,E2 -20860.733} C_VEL
LIN {X 0,Y 215.138,Z 420.004,A -85,B 0,C 180,E1 -20861.488,E2 -20861.488} C_VEL
LIN {X 0,Y 214.549,Z 418.141,A -85,B 0,C 180,E1 -20861.833,E2 -20861.833} C_VEL
LIN {X 0,Y 214.395,Z 416.456,A -85,B 0,C 180,E1 -20866.734,E2 -20866.734} C_VEL
LIN {X 0,Y 214.394,Z 415.338,A -85,B 0,C 180,E1 -20870.566,E2 -20870.566} C_VEL
LIN {X 0,Y 214.391,Z 414.858,A -85,B 0,C 180,E1 -20872.465,E2 -20872.465} C_VEL
LIN {X 0,Y 214.443,Z 413.772,A -85,B 0,C 180,E1 -20878.122,E2 -20878.122} C_VEL
LIN {X 0,Y 214.548,Z 413.755,A -85,B 0,C 180,E1 -20880,E2 -20880} C_VEL
LIN {X 0,Y 214.443,Z 413.769,A -85,B 0,C 180,E1 -20881.878,E2 -20881.878} C_VEL
LIN {X 0,Y 214.196,Z 413.799,A -85,B 0,C 180,E1 -20887.541,E2 -20887.541} C_VEL
LIN {X 0,Y 213.997,Z 413.824,A -85,B 0,C 180,E1 -20891.364,E2 -20891.364} C_VEL
LIN {X 0,Y 213.99,Z 414.078,A -85,B 0,C 180,E1 -20895.233,E2 -20895.233} C_VEL
LIN {X 0,Y 214.054,Z 414.965,A -85,B 0,C 180,E1 -20899.167,E2 -20899.167} C_VEL
LIN {X 0,Y 214.256,Z 416.212,A -85,B 0,C 180,E1 -20903.3,E2 -20903.3} C_VEL
LIN {X 0,Y 214.56,Z 417.988,A -85,B 0,C 180,E1 -20907.824,E2 -20907.824} C_VEL
LIN {X 0,Y 214.869,Z 419.88,A -85,B 0,C 180,E1 -20911.744,E2 -20911.744} C_VEL
LIN {X 0,Y 215.273,Z 422.318,A -85,B 0,C 180,E1 -20915.99,E2 -20915.99} C_VEL
LIN {X 0,Y 215.551,Z 423.93,A -85,B 0,C 180,E1 -20918.509,E2 -20918.509} C_VEL
LIN {X 0,Y 216.083,Z 427.215,A -85,B 0,C 180,E1 -20923.08,E2 -20923.08} C_VEL
LIN {X 0,Y 216.892,Z 431.36,A -85,B 0,C 180,E1 -20928.183,E2 -20928.183} C_VEL
LIN {X 0,Y 217.157,Z 433.718,A -85,B 0,C 180,E1 -20930.812,E2 -20930.812} C_VEL
LIN {X 0,Y 218.221,Z 437.004,A -85,B 0,C 180,E1 -20931.365,E2 -20931.365} C_VEL
LIN {X 0,Y 219.485,Z 439.362,A -85,B 0,C 180,E1 -20931.885,E2 -20931.885} C_VEL
LIN {X 0,Y 222.443,Z 448.504,A -85,B 0,C 180,E1 -20933.435,E2 -20933.435} C_VEL
LIN {X 0,Y 224.932,Z 459.253,A -85,B 0,C 180,E1 -20935.231,E2 -20935.231} C_VEL
LIN {X 0,Y 226.416,Z 469.29,A -85,B 0,C 180,E1 -20936.939,E2 -20936.939} C_VEL
LIN {X 0,Y 227.058,Z 481.29,A -85,B 0,C 180,E1 -20939.108,E2 -20939.108} C_VEL
LIN {X 0,Y 226.593,Z 491.073,A -85,B 0,C 180,E1 -20941.034,E2 -20941.034} C_VEL
LIN {X 0,Y 225.369,Z 500.508,A -85,B 0,C 180,E1 -20943.117,E2 -20943.117} C_VEL
LIN {X 0,Y 224.134,Z 504.879,A -85,B 0,C 180,E1 -20944.134,E2 -20944.134} C_VEL
LIN {X 0,Y 222.178,Z 509.022,A -85,B 0,C 180,E1 -20945.098,E2 -20945.098} C_VEL
LIN {X 0,Y 217.423,Z 515.367,A -85,B 0,C 180,E1 -20946.636,E2 -20946.636} C_VEL
LIN {X 0,Y 212.678,Z 521.137,A -85,B 0,C 180,E1 -20948.361,E2 -20948.361} C_VEL
LIN {X 0,Y 210.778,Z 524.297,A -85,B 0,C 180,E1 -20949.605,E2 -20949.605} C_VEL
LIN {X 0,Y 208.58,Z 529.949,A -85,B 0,C 180,E1 -20952.347,E2 -20952.347} C_VEL
LIN {X 0,Y 206.769,Z 534.612,A -85,B 0,C 180,E1 -20955.231,E2 -20955.231} C_VEL
LIN {X 0,Y 205.57,Z 538.212,A -85,B 0,C 180,E1 -20958.163,E2 -20958.163} C_VEL
LIN {X 0,Y 205.064,Z 540.059,A -85,B 0,C 180,E1 -20960.133,E2 -20960.133} C_VEL
LIN {X 0,Y 204.578,Z 542.535,A -85,B 0,C 180,E1 -20964.084,E2 -20964.084} C_VEL
LIN {X 0,Y 204.555,Z 543.194,A -85,B 0,C 180,E1 -20966.059,E2 -20966.059} C_VEL
LIN {X 0,Y 204.679,Z 543.433,A -85,B 0,C 180,E1 -20968.032,E2 -20968.032} C_VEL
LIN {X 0,Y 204.748,Z 543.248,A -85,B 0,C 180,E1 -20970,E2 -20970} C_VEL
LIN {X 0,Y 204.708,Z 542.657,A -85,B 0,C 180,E1 -20971.967,E2 -20971.967} C_VEL
LIN {X 0,Y 204.714,Z 540.645,A -85,B 0,C 180,E1 -20975.379,E2 -20975.379} C_VEL
LIN {X 0,Y 204.948,Z 537.216,A -85,B 0,C 180,E1 -20978.876,E2 -20978.876} C_VEL
LIN {X 0,Y 205.584,Z 533.138,A -85,B 0,C 180,E1 -20981.835,E2 -20981.835} C_VEL
LIN {X 0,Y 206.944,Z 526.863,A -85,B 0,C 180,E1 -20985.259,E2 -20985.259} C_VEL
LIN {X 0,Y 208.643,Z 520.025,A -85,B 0,C 180,E1 -20988.154,E2 -20988.154} C_VEL
LIN {X 0,Y 210.38,Z 513.036,A -85,B 0,C 180,E1 -20990.535,E2 -20990.535} C_VEL
LIN {X 0,Y 212.435,Z 504.635,A -85,B 0,C 180,E1 -20992.874,E2 -20992.874} C_VEL
LIN {X 0,Y 214.409,Z 496.562,A -85,B 0,C 180,E1 -20994.703,E2 -20994.703} C_VEL
LIN {X 0,Y 214.572,Z 486.493,A -85,B 0,C 180,E1 -20996.766,E2 -20996.766} C_VEL
LIN {X 0,Y 214.197,Z 475.263,A -85,B 0,C 180,E1 -20998.693,E2 -20998.693} C_VEL
LIN {X 0,Y 213.039,Z 463.272,A -85,B 0,C 180,E1 -21000.424,E2 -21000.424} C_VEL
LIN {X 0,Y 211.138,Z 450.207,A -85,B 0,C 180,E1 -21001.99,E2 -21001.99} C_VEL
LIN {X 0,Y 208.354,Z 436.444,A -85,B 0,C 180,E1 -21003.332,E2 -21003.332} C_VEL
LIN {X 0,Y 209.479,Z 432.322,A -85,B 0,C 180,E1 -21007.148,E2 -21007.148} C_VEL
LIN {X 0,Y 209.472,Z 429.803,A -85,B 0,C 180,E1 -21009.602,E2 -21009.602} C_VEL
LIN {X 0,Y 208.78,Z 425.908,A -85,B 0,C 180,E1 -21013.636,E2 -21013.636} C_VEL
LIN {X 0,Y 207.993,Z 421.929,A -85,B 0,C 180,E1 -21018.017,E2 -21018.017} C_VEL
LIN {X 0,Y 207.32,Z 418.188,A -85,B 0,C 180,E1 -21022.397,E2 -21022.397} C_VEL
LIN {X 0,Y 206.751,Z 414.732,A -85,B 0,C 180,E1 -21026.761,E2 -21026.761} C_VEL
LIN {X 0,Y 206.762,Z 414.732,A -85,B 0,C 180,E1 -21032.096,E2 -21032.096} C_VEL
LIN {X 0,Y 206.781,Z 414.728,A -85,B 0,C 180,E1 -21036.583,E2 -21036.583} C_VEL
LIN {X 0,Y 206.872,Z 414.715,A -85,B 0,C 180,E1 -21042.197,E2 -21042.197} C_VEL
LIN {X 0,Y 206.89,Z 414.714,A -85,B 0,C 180,E1 -21046.244,E2 -21046.244} C_VEL
LIN {X 0,Y 207.094,Z 414.688,A -85,B 0,C 180,E1 -21050.231,E2 -21050.231} C_VEL
LIN {X 0,Y 207.056,Z 414.684,A -85,B 0,C 180,E1 -21054.156,E2 -21054.156} C_VEL
LIN {X 0,Y 207.376,Z 414.652,A -85,B 0,C 180,E1 -21058.058,E2 -21058.058} C_VEL
LIN {X 0,Y 207.513,Z 414.635,A -85,B 0,C 180,E1 -21060,E2 -21060} C_VEL
LIN {X 0,Y 207.079,Z 414.678,A -85,B 0,C 180,E1 -21063.892,E2 -21063.892} C_VEL
LIN {X 0,Y 207.163,Z 414.678,A -85,B 0,C 180,E1 -21067.799,E2 -21067.799} C_VEL
LIN {X 0,Y 206.976,Z 414.696,A -85,B 0,C 180,E1 -21071.756,E2 -21071.756} C_VEL
LIN {X 0,Y 206.861,Z 414.713,A -85,B 0,C 180,E1 -21075.771,E2 -21075.771} C_VEL
LIN {X 0,Y 206.779,Z 414.726,A -85,B 0,C 180,E1 -21079.87,E2 -21079.87} C_VEL
LIN {X 0,Y 206.76,Z 414.72,A -85,B 0,C 180,E1 -21084.073,E2 -21084.073} C_VEL
LIN {X 0,Y 206.741,Z 414.733,A -85,B 0,C 180,E1 -21088.42,E2 -21088.42} C_VEL
LIN {X 0,Y 206.706,Z 414.728,A -85,B 0,C 180,E1 -21092.957,E2 -21092.957} C_VEL
LIN {X 0,Y 206.719,Z 414.732,A -85,B 0,C 180,E1 -21095.321,E2 -21095.321} C_VEL
LIN {X 0,Y 206.669,Z 414.734,A -85,B 0,C 180,E1 -21100.25,E2 -21100.25} C_VEL
LIN {X 0,Y 206.647,Z 414.746,A -85,B 0,C 180,E1 -21104.424,E2 -21104.424} C_VEL
LIN {X 0,Y 206.659,Z 414.728,A -85,B 0,C 180,E1 -21109.75,E2 -21109.75} C_VEL
LIN {X 0,Y 206.699,Z 414.724,A -85,B 0,C 180,E1 -21114.69,E2 -21114.69} C_VEL
LIN {X 0,Y 206.707,Z 414.739,A -85,B 0,C 180,E1 -21119.338,E2 -21119.338} C_VEL
LIN {X 0,Y 206.733,Z 414.717,A -85,B 0,C 180,E1 -21123.773,E2 -21123.773} C_VEL
LIN {X 0,Y 206.76,Z 414.731,A -85,B 0,C 180,E1 -21128.044,E2 -21128.044} C_VEL
LIN {X 0,Y 206.875,Z 414.704,A -85,B 0,C 180,E1 -21132.198,E2 -21132.198} C_VEL
LIN {X 0,Y 206.917,Z 414.712,A -85,B 0,C 180,E1 -21136.247,E2 -21136.247} C_VEL
LIN {X 0,Y 207.136,Z 414.68,A -85,B 0,C 180,E1 -21140.233,E2 -21140.233} C_VEL
LIN {X 0,Y 207.19,Z 414.678,A -85,B 0,C 180,E1 -21142.203,E2 -21142.203} C_VEL
LIN {X 0,Y 207.234,Z 414.672,A -85,B 0,C 180,E1 -21148.057,E2 -21148.057} C_VEL
LIN {X 0,Y 206.918,Z 414.711,A -85,B 0,C 180,E1 -21148.784,E2 -21148.784} C_VEL
LIN {X 0,Y 210.418,Z 425.72,A -85,B 0,C 180,E1 -21150.101,E2 -21150.101} C_VEL
LIN {X 0,Y 213.471,Z 434.834,A -85,B 0,C 180,E1 -21151.415,E2 -21151.415} C_VEL
LIN {X 0,Y 216.111,Z 446.093,A -85,B 0,C 180,E1 -21153.147,E2 -21153.147} C_VEL
LIN {X 0,Y 218.055,Z 457.035,A -85,B 0,C 180,E1 -21155.085,E2 -21155.085} C_VEL
LIN {X 0,Y 218.372,Z 459.38,A -85,B 0,C 180,E1 -21155.541,E2 -21155.541} C_VEL
LIN {X 0,Y 216.212,Z 470.191,A -85,B 0,C 180,E1 -21157.471,E2 -21157.471} C_VEL
LIN {X 0,Y 213.895,Z 480.07,A -85,B 0,C 180,E1 -21159.693,E2 -21159.693} C_VEL
LIN {X 0,Y 211.455,Z 489.869,A -85,B 0,C 180,E1 -21162.477,E2 -21162.477} C_VEL
LIN {X 0,Y 209.499,Z 497.395,A -85,B 0,C 180,E1 -21165.178,E2 -21165.178} C_VEL
LIN {X 0,Y 208.023,Z 503.065,A -85,B 0,C 180,E1 -21167.702,E2 -21167.702} C_VEL
LIN {X 0,Y 206.556,Z 508.766,A -85,B 0,C 180,E1 -21170.932,E2 -21170.932} C_VEL
LIN {X 0,Y 205.597,Z 513.098,A -85,B 0,C 180,E1 -21174.217,E2 -21174.217} C_VEL
LIN {X 0,Y 204.962,Z 515.712,A -85,B 0,C 180,E1 -21176.934,E2 -21176.934} C_VEL
LIN {X 0,Y 204.574,Z 518.039,A -85,B 0,C 180,E1 -21180.81,E2 -21180.81} C_VEL
LIN {X 0,Y 204.669,Z 518.809,A -85,B 0,C 180,E1 -21184.5,E2 -21184.5} C_VEL
LIN {X 0,Y 205.316,Z 518.212,A -85,B 0,C 180,E1 -21188.066,E2 -21188.066} C_VEL
LIN {X 0,Y 206.44,Z 516.403,A -85,B 0,C 180,E1 -21191.499,E2 -21191.499} C_VEL
LIN {X 0,Y 208.083,Z 513.057,A -85,B 0,C 180,E1 -21195.175,E2 -21195.175} C_VEL
LIN {X 0,Y 210.439,Z 507.957,A -85,B 0,C 180,E1 -21198.837,E2 -21198.837} C_VEL
LIN {X 0,Y 212.72,Z 502.894,A -85,B 0,C 180,E1 -21201.536,E2 -21201.536} C_VEL
LIN {X 0,Y 215.736,Z 495.695,A -85,B 0,C 180,E1 -21204.529,E2 -21204.529} C_VEL
LIN {X 0,Y 219.112,Z 486.831,A -85,B 0,C 180,E1 -21207.346,E2 -21207.346} C_VEL
LIN {X 0,Y 222.255,Z 477.806,A -85,B 0,C 180,E1 -21209.606,E2 -21209.606} C_VEL
LIN {X 0,Y 224.975,Z 468.48,A -85,B 0,C 180,E1 -21211.506,E2 -21211.506} C_VEL
LIN {X 0,Y 224.182,Z 460.309,A -85,B 0,C 180,E1 -21213.465,E2 -21213.465} C_VEL
LIN {X 0,Y 222.2,Z 450.718,A -85,B 0,C 180,E1 -21215.721,E2 -21215.721} C_VEL
LIN {X 0,Y 219.236,Z 441.372,A -85,B 0,C 180,E1 -21217.934,E2 -21217.934} C_VEL
LIN {X 0,Y 214.783,Z 431.549,A -85,B 0,C 180,E1 -21220.442,E2 -21220.442} C_VEL
LIN {X 0,Y 212.404,Z 427.307,A -85,B 0,C 180,E1 -21221.62,E2 -21221.62} C_VEL
LIN {X 0,Y 210.705,Z 424.19,A -85,B 0,C 180,E1 -21222.469,E2 -21222.469} C_VEL
LIN {X 0,Y 208.14,Z 420.72,A -85,B 0,C 180,E1 -21223.636,E2 -21223.636} C_VEL
LIN {X 0,Y 207.507,Z 418.832,A -85,B 0,C 180,E1 -21224.027,E2 -21224.027} C_VEL
LIN {X 0,Y 207.453,Z 417.262,A -85,B 0,C 180,E1 -21229.246,E2 -21229.246} C_VEL
LIN {X 0,Y 207.475,Z 416.518,A -85,B 0,C 180,E1 -21232.212,E2 -21232.212} C_VEL
LIN {X 0,Y 207.517,Z 415.435,A -85,B 0,C 180,E1 -21238.059,E2 -21238.059} C_VEL
LIN {X 0,Y 207.614,Z 415.172,A -85,B 0,C 180,E1 -21240,E2 -21240} C_VEL
LIN {X 0,Y 207.137,Z 415.02,A -85,B 0,C 180,E1 -21243.891,E2 -21243.891} C_VEL
LIN {X 0,Y 207.18,Z 415.019,A -85,B 0,C 180,E1 -21247.798,E2 -21247.798} C_VEL
LIN {X 0,Y 207.053,Z 415.344,A -85,B 0,C 180,E1 -21251.751,E2 -21251.751} C_VEL
LIN {X 0,Y 207.117,Z 415.943,A -85,B 0,C 180,E1 -21255.751,E2 -21255.751} C_VEL
LIN {X 0,Y 207.19,Z 416.897,A -85,B 0,C 180,E1 -21259.828,E2 -21259.828} C_VEL
LIN {X 0,Y 207.377,Z 418.193,A -85,B 0,C 180,E1 -21263.996,E2 -21263.996} C_VEL
LIN {X 0,Y 207.701,Z 419.934,A -85,B 0,C 180,E1 -21268.387,E2 -21268.387} C_VEL
LIN {X 0,Y 208.017,Z 422.063,A -85,B 0,C 180,E1 -21272.722,E2 -21272.722} C_VEL
LIN {X 0,Y 208.357,Z 423.874,A -85,B 0,C 180,E1 -21275.95,E2 -21275.95} C_VEL
LIN {X 0,Y 208.747,Z 426.302,A -85,B 0,C 180,E1 -21279.768,E2 -21279.768} C_VEL
LIN {X 0,Y 209.043,Z 428.077,A -85,B 0,C 180,E1 -21282.3,E2 -21282.3} C_VEL
LIN {X 0,Y 209.799,Z 432.066,A -85,B 0,C 180,E1 -21287.474,E2 -21287.474} C_VEL
LIN {X 0,Y 209.982,Z 433.069,A -85,B 0,C 180,E1 -21288.681,E2 -21288.681} C_VEL
LIN {X 0,Y 211.142,Z 436.328,A -85,B 0,C 180,E1 -21289.298,E2 -21289.298} C_VEL
LIN {X 0,Y 212.876,Z 439.193,A -85,B 0,C 180,E1 -21290.052,E2 -21290.052} C_VEL
LIN {X 0,Y 215.12,Z 444.751,A -85,B 0,C 180,E1 -21291.208,E2 -21291.208} C_VEL
LIN {X 0,Y 217.136,Z 451.421,A -85,B 0,C 180,E1 -21292.464,E2 -21292.464} C_VEL
LIN {X 0,Y 219.325,Z 461.954,A -85,B 0,C 180,E1 -21294.357,E2 -21294.357} C_VEL
LIN {X 0,Y 220.537,Z 472.301,A -85,B 0,C 180,E1 -21296.258,E2 -21296.258} C_VEL
LIN {X 0,Y 220.879,Z 483.547,A -85,B 0,C 180,E1 -21298.439,E2 -21298.439} C_VEL
LIN {X 0,Y 220.114,Z 493.566,A -85,B 0,C 180,E1 -21300.545,E2 -21300.545} C_VEL
LIN {X 0,Y 218.583,Z 502.757,A -85,B 0,C 180,E1 -21302.731,E2 -21302.731} C_VEL
LIN {X 0,Y 214.968,Z 512.627,A -85,B 0,C 180,E1 -21305.365,E2 -21305.365} C_VEL
LIN {X 0,Y 211.942,Z 520.91,A -85,B 0,C 180,E1 -21308.199,E2 -21308.199} C_VEL
LIN {X 0,Y 210.778,Z 524.297,A -85,B 0,C 180,E1 -21309.605,E2 -21309.605} C_VEL
LIN {X 0,Y 208.914,Z 527.293,A -85,B 0,C 180,E1 -21310.915,E2 -21310.915} C_VEL
LIN {X 0,Y 202.535,Z 533.138,A -85,B 0,C 180,E1 -21313.942,E2 -21313.942} C_VEL
LIN {X 0,Y 199.597,Z 535.884,A -85,B 0,C 180,E1 -21315.877,E2 -21315.877} C_VEL
LIN {X 0,Y 198.864,Z 537.085,A -85,B 0,C 180,E1 -21316.93,E2 -21316.93} C_VEL
LIN {X 0,Y 198.03,Z 539.756,A -85,B 0,C 180,E1 -21319.779,E2 -21319.779} C_VEL
LIN {X 0,Y 197.501,Z 542.173,A -85,B 0,C 180,E1 -21323.871,E2 -21323.871} C_VEL
LIN {X 0,Y 197.463,Z 542.791,A -85,B 0,C 180,E1 -21325.918,E2 -21325.918} C_VEL
LIN {X 0,Y 197.586,Z 542.982,A -85,B 0,C 180,E1 -21327.961,E2 -21327.961} C_VEL
LIN {X 0,Y 197.68,Z 542.771,A -85,B 0,C 180,E1 -21329.999,E2 -21329.999} C_VEL
LIN {X 0,Y 197.642,Z 542.153,A -85,B 0,C 180,E1 -21332.037,E2 -21332.037} C_VEL
LIN {X 0,Y 197.622,Z 540.289,A -85,B 0,C 180,E1 -21335.278,E2 -21335.278} C_VEL
LIN {X 0,Y 197.919,Z 536.562,A -85,B 0,C 180,E1 -21339.194,E2 -21339.194} C_VEL
LIN {X 0,Y 198.596,Z 532.417,A -85,B 0,C 180,E1 -21342.258,E2 -21342.258} C_VEL
LIN {X 0,Y 200.092,Z 526.075,A -85,B 0,C 180,E1 -21345.795,E2 -21345.795} C_VEL
LIN {X 0,Y 201.886,Z 519.156,A -85,B 0,C 180,E1 -21348.784,E2 -21348.784} C_VEL
LIN {X 0,Y 203.997,Z 511.1,A -85,B 0,C 180,E1 -21351.535,E2 -21351.535} C_VEL
LIN {X 0,Y 206.358,Z 501.585,A -85,B 0,C 180,E1 -21354.121,E2 -21354.121} C_VEL
LIN {X 0,Y 207.579,Z 496.416,A -85,B 0,C 180,E1 -21355.304,E2 -21355.304} C_VEL
LIN {X 0,Y 207.749,Z 486.353,A -85,B 0,C 180,E1 -21357.446,E2 -21357.446} C_VEL
LIN {X 0,Y 207.406,Z 475.277,A -85,B 0,C 180,E1 -21359.426,E2 -21359.426} C_VEL
LIN {X 0,Y 206.205,Z 462.397,A -85,B 0,C 180,E1 -21361.359,E2 -21361.359} C_VEL
LIN {X 0,Y 204.317,Z 449.493,A -85,B 0,C 180,E1 -21362.97,E2 -21362.97} C_VEL
LIN {X 0,Y 201.57,Z 436.022,A -85,B 0,C 180,E1 -21364.359,E2 -21364.359} C_VEL
LIN {X 0,Y 202.359,Z 433.277,A -85,B 0,C 180,E1 -21366.984,E2 -21366.984} C_VEL
LIN {X 0,Y 202.492,Z 431.6,A -85,B 0,C 180,E1 -21368.661,E2 -21368.661} C_VEL
LIN {X 0,Y 202.169,Z 429.034,A -85,B 0,C 180,E1 -21371.336,E2 -21371.336} C_VEL
LIN {X 0,Y 201.365,Z 425.049,A -85,B 0,C 180,E1 -21375.73,E2 -21375.73} C_VEL
LIN {X 0,Y 200.543,Z 420.661,A -85,B 0,C 180,E1 -21380.89,E2 -21380.89} C_VEL
LIN {X 0,Y 199.922,Z 416.81,A -85,B 0,C 180,E1 -21385.774,E2 -21385.774} C_VEL
LIN {X 0,Y 199.683,Z 415.615,A -85,B 0,C 180,E1 -21387.637,E2 -21387.637} C_VEL
LIN {X 0,Y 199.683,Z 415.615,A -85,B 0,C 180,E1 -21392.771,E2 -21392.771} C_VEL
LIN {X 0,Y 199.733,Z 415.606,A -85,B 0,C 180,E1 -21397.229,E2 -21397.229} C_VEL
LIN {X 0,Y 199.833,Z 415.592,A -85,B 0,C 180,E1 -21401.722,E2 -21401.722} C_VEL
LIN {X 0,Y 199.831,Z 415.592,A -85,B 0,C 180,E1 -21405.748,E2 -21405.748} C_VEL
LIN {X 0,Y 200.018,Z 415.569,A -85,B 0,C 180,E1 -21409.882,E2 -21409.882} C_VEL
LIN {X 0,Y 200.018,Z 415.561,A -85,B 0,C 180,E1 -21413.949,E2 -21413.949} C_VEL
LIN {X 0,Y 200.316,Z 415.531,A -85,B 0,C 180,E1 -21417.99,E2 -21417.99} C_VEL
LIN {X 0,Y 200.477,Z 415.511,A -85,B 0,C 180,E1 -21420,E2 -21420} C_VEL
LIN {X 0,Y 200.025,Z 415.557,A -85,B 0,C 180,E1 -21424.03,E2 -21424.03} C_VEL
LIN {X 0,Y 200.106,Z 415.558,A -85,B 0,C 180,E1 -21428.076,E2 -21428.076} C_VEL
LIN {X 0,Y 199.908,Z 415.573,A -85,B 0,C 180,E1 -21432.178,E2 -21432.178} C_VEL
LIN {X 0,Y 199.799,Z 415.595,A -85,B 0,C 180,E1 -21436.344,E2 -21436.344} C_VEL
LIN {X 0,Y 199.696,Z 415.605,A -85,B 0,C 180,E1 -21440.606,E2 -21440.606} C_VEL
LIN {X 0,Y 199.669,Z 415.609,A -85,B 0,C 180,E1 -21444.985,E2 -21444.985} C_VEL
LIN {X 0,Y 199.672,Z 415.61,A -85,B 0,C 180,E1 -21449.523,E2 -21449.523} C_VEL
LIN {X 0,Y 199.661,Z 415.604,A -85,B 0,C 180,E1 -21452.353,E2 -21452.353} C_VEL
LIN {X 0,Y 199.638,Z 415.617,A -85,B 0,C 180,E1 -21456.76,E2 -21456.76} C_VEL
LIN {X 0,Y 199.638,Z 415.613,A -85,B 0,C 180,E1 -21459.322,E2 -21459.322} C_VEL
LIN {X 0,Y 199.588,Z 415.617,A -85,B 0,C 180,E1 -21462.316,E2 -21462.316} C_VEL
LIN {X 0,Y 199.586,Z 415.623,A -85,B 0,C 180,E1 -21465.232,E2 -21465.232} C_VEL
LIN {X 0,Y 199.578,Z 415.619,A -85,B 0,C 180,E1 -21468.006,E2 -21468.006} C_VEL
LIN {X 0,Y 199.608,Z 415.599,A -85,B 0,C 180,E1 -21470.769,E2 -21470.769} C_VEL
LIN {X 0,Y 199.611,Z 415.613,A -85,B 0,C 180,E1 -21475.715,E2 -21475.715} C_VEL
LIN {X 0,Y 199.693,Z 415.614,A -85,B 0,C 180,E1 -21478.137,E2 -21478.137} C_VEL
LIN {X 0,Y 199.686,Z 415.601,A -85,B 0,C 180,E1 -21482.773,E2 -21482.773} C_VEL
LIN {X 0,Y 199.74,Z 415.6,A -85,B 0,C 180,E1 -21487.23,E2 -21487.23} C_VEL
LIN {X 0,Y 199.798,Z 415.587,A -85,B 0,C 180,E1 -21491.758,E2 -21491.758} C_VEL
LIN {X 0,Y 199.851,Z 415.592,A -85,B 0,C 180,E1 -21495.75,E2 -21495.75} C_VEL
LIN {X 0,Y 200.078,Z 415.556,A -85,B 0,C 180,E1 -21499.885,E2 -21499.885} C_VEL
LIN {X 0,Y 200.134,Z 415.558,A -85,B 0,C 180,E1 -21501.926,E2 -21501.926} C_VEL
LIN {X 0,Y 200.139,Z 415.556,A -85,B 0,C 180,E1 -21507.799,E2 -21507.799} C_VEL
LIN {X 0,Y 204.404,Z 428.823,A -85,B 0,C 180,E1 -21509.521,E2 -21509.521} C_VEL
LIN {X 0,Y 207.406,Z 438.263,A -85,B 0,C 180,E1 -21510.97,E2 -21510.97} C_VEL
LIN {X 0,Y 209.746,Z 448.748,A -85,B 0,C 180,E1 -21512.711,E2 -21512.711} C_VEL
LIN {X 0,Y 211.645,Z 460.732,A -85,B 0,C 180,E1 -21514.992,E2 -21514.992} C_VEL
LIN {X 0,Y 209.389,Z 471.389,A -85,B 0,C 180,E1 -21516.989,E2 -21516.989} C_VEL
LIN {X 0,Y 207.073,Z 480.779,A -85,B 0,C 180,E1 -21519.185,E2 -21519.185} C_VEL
LIN {X 0,Y 204.689,Z 490.016,A -85,B 0,C 180,E1 -21521.889,E2 -21521.889} C_VEL
LIN {X 0,Y 202.749,Z 497.178,A -85,B 0,C 180,E1 -21524.504,E2 -21524.504} C_VEL
LIN {X 0,Y 201.083,Z 503.314,A -85,B 0,C 180,E1 -21527.283,E2 -21527.283} C_VEL
LIN {X 0,Y 199.546,Z 509.066,A -85,B 0,C 180,E1 -21530.622,E2 -21530.622} C_VEL
LIN {X 0,Y 198.525,Z 513.49,A -85,B 0,C 180,E1 -21534.074,E2 -21534.074} C_VEL
LIN {X 0,Y 197.773,Z 516.59,A -85,B 0,C 180,E1 -21537.514,E2 -21537.514} C_VEL
LIN {X 0,Y 197.476,Z 518.633,A -85,B 0,C 180,E1 -21541.334,E2 -21541.334} C_VEL
LIN {X 0,Y 197.673,Z 519.239,A -85,B 0,C 180,E1 -21545.141,E2 -21545.141} C_VEL
LIN {X 0,Y 198.42,Z 518.543,A -85,B 0,C 180,E1 -21548.809,E2 -21548.809} C_VEL
LIN {X 0,Y 199.657,Z 516.65,A -85,B 0,C 180,E1 -21552.335,E2 -21552.335} C_VEL
LIN {X 0,Y 201.227,Z 513.657,A -85,B 0,C 180,E1 -21555.691,E2 -21555.691} C_VEL
LIN {X 0,Y 203.671,Z 508.746,A -85,B 0,C 180,E1 -21559.388,E2 -21559.388} C_VEL
LIN {X 0,Y 206.042,Z 503.863,A -85,B 0,C 180,E1 -21562.122,E2 -21562.122} C_VEL
LIN {X 0,Y 209.129,Z 496.923,A -85,B 0,C 180,E1 -21565.158,E2 -21565.158} C_VEL
LIN {X 0,Y 212.078,Z 489.854,A -85,B 0,C 180,E1 -21567.584,E2 -21567.584} C_VEL
LIN {X 0,Y 215.248,Z 481.437,A -85,B 0,C 180,E1 -21569.91,E2 -21569.91} C_VEL
LIN {X 0,Y 218.628,Z 471.226,A -85,B 0,C 180,E1 -21572.129,E2 -21572.129} C_VEL
LIN {X 0,Y 218.833,Z 470.416,A -85,B 0,C 180,E1 -21572.293,E2 -21572.293} C_VEL
LIN {X 0,Y 217.923,Z 460.842,A -85,B 0,C 180,E1 -21574.753,E2 -21574.753} C_VEL
LIN {X 0,Y 216.05,Z 451.821,A -85,B 0,C 180,E1 -21577.023,E2 -21577.023} C_VEL
LIN {X 0,Y 213.291,Z 443.164,A -85,B 0,C 180,E1 -21579.254,E2 -21579.254} C_VEL
LIN {X 0,Y 208.66,Z 433.093,A -85,B 0,C 180,E1 -21582.095,E2 -21582.095} C_VEL
LIN {X 0,Y 206.696,Z 429.558,A -85,B 0,C 180,E1 -21583.201,E2 -21583.201} C_VEL
LIN {X 0,Y 204.157,Z 425.57,A -85,B 0,C 180,E1 -21584.552,E2 -21584.552} C_VEL
LIN {X 0,Y 203.348,Z 424.294,A -85,B 0,C 180,E1 -21584.975,E2 -21584.975} C_VEL
LIN {X 0,Y 201.335,Z 421.823,A -85,B 0,C 180,E1 -21585.985,E2 -21585.985} C_VEL
LIN {X 0,Y 200.511,Z 419.554,A -85,B 0,C 180,E1 -21586.573,E2 -21586.573} C_VEL
LIN {X 0,Y 200.525,Z 418.655,A -85,B 0,C 180,E1 -21589.907,E2 -21589.907} C_VEL
LIN {X 0,Y 200.551,Z 418.19,A -85,B 0,C 180,E1 -21591.942,E2 -21591.942} C_VEL
LIN {X 0,Y 200.616,Z 417.113,A -85,B 0,C 180,E1 -21597.992,E2 -21597.992} C_VEL
LIN {X 0,Y 200.722,Z 416.863,A -85,B 0,C 180,E1 -21600,E2 -21600} C_VEL
LIN {X 0,Y 200.262,Z 416.732,A -85,B 0,C 180,E1 -21604.025,E2 -21604.025} C_VEL
LIN {X 0,Y 200.294,Z 416.795,A -85,B 0,C 180,E1 -21608.068,E2 -21608.068} C_VEL
LIN {X 0,Y 200.182,Z 417.153,A -85,B 0,C 180,E1 -21612.16,E2 -21612.16} C_VEL
LIN {X 0,Y 200.25,Z 417.816,A -85,B 0,C 180,E1 -21616.306,E2 -21616.306} C_VEL
LIN {X 0,Y 200.313,Z 418.859,A -85,B 0,C 180,E1 -21620.539,E2 -21620.539} C_VEL
LIN {X 0,Y 200.517,Z 420.252,A -85,B 0,C 180,E1 -21624.872,E2 -21624.872} C_VEL
LIN {X 0,Y 200.834,Z 422.062,A -85,B 0,C 180,E1 -21629.335,E2 -21629.335} C_VEL
LIN {X 0,Y 201.219,Z 424.351,A -85,B 0,C 180,E1 -21633.975,E2 -21633.975} C_VEL
LIN {X 0,Y 201.487,Z 425.87,A -85,B 0,C 180,E1 -21636.655,E2 -21636.655} C_VEL
LIN {X 0,Y 201.938,Z 428.916,A -85,B 0,C 180,E1 -21641.395,E2 -21641.395} C_VEL
LIN {X 0,Y 202.618,Z 432.52,A -85,B 0,C 180,E1 -21646.162,E2 -21646.162} C_VEL
LIN {X 0,Y 203.712,Z 435.46,A -85,B 0,C 180,E1 -21646.8,E2 -21646.8} C_VEL
LIN {X 0,Y 206.022,Z 438.757,A -85,B 0,C 180,E1 -21647.899,E2 -21647.899} C_VEL
LIN {X 0,Y 207.967,Z 442.954,A -85,B 0,C 180,E1 -21648.957,E2 -21648.957} C_VEL
LIN {X 0,Y 210.409,Z 449.071,A -85,B 0,C 180,E1 -21650.372,E2 -21650.372} C_VEL
LIN {X 0,Y 212.51,Z 457.456,A -85,B 0,C 180,E1 -21652.046,E2 -21652.046} C_VEL
LIN {X 0,Y 214.238,Z 468.967,A -85,B 0,C 180,E1 -21654.289,E2 -21654.289} C_VEL
LIN {X 0,Y 214.777,Z 479.885,A -85,B 0,C 180,E1 -21656.483,E2 -21656.483} C_VEL
LIN {X 0,Y 214.343,Z 489.944,A -85,B 0,C 180,E1 -21658.659,E2 -21658.659} C_VEL
LIN {X 0,Y 212.999,Z 499.341,A -85,B 0,C 180,E1 -21660.877,E2 -21660.877} C_VEL
LIN {X 0,Y 211.675,Z 504.843,A -85,B 0,C 180,E1 -21662.301,E2 -21662.301} C_VEL
LIN {X 0,Y 208.537,Z 512.818,A -85,B 0,C 180,E1 -21664.552,E2 -21664.552} C_VEL
LIN {X 0,Y 205.918,Z 519.491,A -85,B 0,C 180,E1 -21666.891,E2 -21666.891} C_VEL
LIN {X 0,Y 203.302,Z 526.119,A -85,B 0,C 180,E1 -21669.776,E2 -21669.776} C_VEL
LIN {X 0,Y 201.09,Z 531.467,A -85,B 0,C 180,E1 -21672.718,E2 -21672.718} C_VEL
LIN {X 0,Y 199.338,Z 535.693,A -85,B 0,C 180,E1 -21675.712,E2 -21675.712} C_VEL
LIN {X 0,Y 198.864,Z 537.085,A -85,B 0,C 180,E1 -21676.93,E2 -21676.93} C_VEL
LIN {X 0,Y 197.672,Z 538.723,A -85,B 0,C 180,E1 -21678.537,E2 -21678.537} C_VEL
LIN {X 0,Y 194.189,Z 540.706,A -85,B 0,C 180,E1 -21681.19,E2 -21681.19} C_VEL
LIN {X 0,Y 191.514,Z 541.755,A -85,B 0,C 180,E1 -21683.399,E2 -21683.399} C_VEL
LIN {X 0,Y 190.443,Z 542.254,A -85,B 0,C 180,E1 -21685.144,E2 -21685.144} C_VEL
LIN {X 0,Y 190.383,Z 542.368,A -85,B 0,C 180,E1 -21685.738,E2 -21685.738} C_VEL
LIN {X 0,Y 190.495,Z 542.529,A -85,B 0,C 180,E1 -21687.885,E2 -21687.885} C_VEL
LIN {X 0,Y 190.613,Z 542.291,A -85,B 0,C 180,E1 -21689.999,E2 -21689.999} C_VEL
LIN {X 0,Y 190.554,Z 541.641,A -85,B 0,C 180,E1 -21692.113,E2 -21692.113} C_VEL
LIN {X 0,Y 190.529,Z 539.925,A -85,B 0,C 180,E1 -21695.163,E2 -21695.163} C_VEL
LIN {X 0,Y 190.885,Z 535.885,A -85,B 0,C 180,E1 -21699.536,E2 -21699.536} C_VEL
LIN {X 0,Y 191.625,Z 531.667,A -85,B 0,C 180,E1 -21702.711,E2 -21702.711} C_VEL
LIN {X 0,Y 192.927,Z 526.257,A -85,B 0,C 180,E1 -21705.855,E2 -21705.855} C_VEL
LIN {X 0,Y 194.749,Z 519.475,A -85,B 0,C 180,E1 -21708.952,E2 -21708.952} C_VEL
LIN {X 0,Y 196.544,Z 512.746,A -85,B 0,C 180,E1 -21711.428,E2 -21711.428} C_VEL
LIN {X 0,Y 198.841,Z 504.222,A -85,B 0,C 180,E1 -21713.982,E2 -21713.982} C_VEL
LIN {X 0,Y 200.75,Z 496.196,A -85,B 0,C 180,E1 -21715.95,E2 -21715.95} C_VEL
LIN {X 0,Y 200.989,Z 485.8,A -85,B 0,C 180,E1 -21718.245,E2 -21718.245} C_VEL
LIN {X 0,Y 200.654,Z 475.292,A -85,B 0,C 180,E1 -21720.208,E2 -21720.208} C_VEL
LIN {X 0,Y 199.654,Z 463.623,A -85,B 0,C 180,E1 -21722.058,E2 -21722.058} C_VEL
LIN {X 0,Y 197.797,Z 450.505,A -85,B 0,C 180,E1 -21723.794,E2 -21723.794} C_VEL
LIN {X 0,Y 195.019,Z 437.348,A -85,B 0,C 180,E1 -21725.259,E2 -21725.259} C_VEL
LIN {X 0,Y 194.789,Z 435.637,A -85,B 0,C 180,E1 -21725.416,E2 -21725.416} C_VEL
LIN {X 0,Y 195.352,Z 433.367,A -85,B 0,C 180,E1 -21727.703,E2 -21727.703} C_VEL
LIN {X 0,Y 195.254,Z 430.831,A -85,B 0,C 180,E1 -21730.381,E2 -21730.381} C_VEL
LIN {X 0,Y 194.427,Z 426.558,A -85,B 0,C 180,E1 -21735.177,E2 -21735.177} C_VEL
LIN {X 0,Y 193.726,Z 422.853,A -85,B 0,C 180,E1 -21739.624,E2 -21739.624} C_VEL
LIN {X 0,Y 193.083,Z 419.148,A -85,B 0,C 180,E1 -21744.382,E2 -21744.382} C_VEL
LIN {X 0,Y 192.662,Z 416.488,A -85,B 0,C 180,E1 -21748.123,E2 -21748.123} C_VEL
LIN {X 0,Y 192.661,Z 416.489,A -85,B 0,C 180,E1 -21751.691,E2 -21751.691} C_VEL
LIN {X 0,Y 192.701,Z 416.481,A -85,B 0,C 180,E1 -21756.348,E2 -21756.348} C_VEL
LIN {X 0,Y 192.777,Z 416.471,A -85,B 0,C 180,E1 -21761.414,E2 -21761.414} C_VEL
LIN {X 0,Y 192.759,Z 416.474,A -85,B 0,C 180,E1 -21765.214,E2 -21765.214} C_VEL
LIN {X 0,Y 192.94,Z 416.45,A -85,B 0,C 180,E1 -21769.567,E2 -21769.567} C_VEL
LIN {X 0,Y 192.98,Z 416.437,A -85,B 0,C 180,E1 -21773.728,E2 -21773.728} C_VEL
LIN {X 0,Y 193.258,Z 416.41,A -85,B 0,C 180,E1 -21777.916,E2 -21777.916} C_VEL
LIN {X 0,Y 193.441,Z 416.388,A -85,B 0,C 180,E1 -21780,E2 -21780} C_VEL
LIN {X 0,Y 192.972,Z 416.436,A -85,B 0,C 180,E1 -21784.177,E2 -21784.177} C_VEL
LIN {X 0,Y 193.057,Z 416.438,A -85,B 0,C 180,E1 -21788.373,E2 -21788.373} C_VEL
LIN {X 0,Y 192.848,Z 416.45,A -85,B 0,C 180,E1 -21792.631,E2 -21792.631} C_VEL
LIN {X 0,Y 192.753,Z 416.474,A -85,B 0,C 180,E1 -21796.959,E2 -21796.959} C_VEL
LIN {X 0,Y 192.632,Z 416.482,A -85,B 0,C 180,E1 -21801.398,E2 -21801.398} C_VEL
LIN {X 0,Y 192.66,Z 416.476,A -85,B 0,C 180,E1 -21804.225,E2 -21804.225} C_VEL
LIN {X 0,Y 192.647,Z 416.486,A -85,B 0,C 180,E1 -21808.893,E2 -21808.893} C_VEL
LIN {X 0,Y 192.597,Z 416.485,A -85,B 0,C 180,E1 -21813.186,E2 -21813.186} C_VEL
LIN {X 0,Y 192.607,Z 416.493,A -85,B 0,C 180,E1 -21816.609,E2 -21816.609} C_VEL
LIN {X 0,Y 192.528,Z 416.491,A -85,B 0,C 180,E1 -21821.077,E2 -21821.077} C_VEL
LIN {X 0,Y 192.516,Z 416.506,A -85,B 0,C 180,E1 -21826.085,E2 -21826.085} C_VEL
LIN {X 0,Y 192.516,Z 416.485,A -85,B 0,C 180,E1 -21830.053,E2 -21830.053} C_VEL
LIN {X 0,Y 192.559,Z 416.478,A -85,B 0,C 180,E1 -21834.271,E2 -21834.271} C_VEL
LIN {X 0,Y 192.607,Z 416.493,A -85,B 0,C 180,E1 -21837.061,E2 -21837.061} C_VEL
LIN {X 0,Y 192.661,Z 416.482,A -85,B 0,C 180,E1 -21841.693,E2 -21841.693} C_VEL
LIN {X 0,Y 192.707,Z 416.471,A -85,B 0,C 180,E1 -21846.35,E2 -21846.35} C_VEL
LIN {X 0,Y 192.734,Z 416.469,A -85,B 0,C 180,E1 -21851.458,E2 -21851.458} C_VEL
LIN {X 0,Y 192.775,Z 416.471,A -85,B 0,C 180,E1 -21855.215,E2 -21855.215} C_VEL
LIN {X 0,Y 193.023,Z 416.433,A -85,B 0,C 180,E1 -21859.511,E2 -21859.511} C_VEL
LIN {X 0,Y 193.081,Z 416.437,A -85,B 0,C 180,E1 -21861.629,E2 -21861.629} C_VEL
LIN {X 0,Y 192.937,Z 416.452,A -85,B 0,C 180,E1 -21866.672,E2 -21866.672} C_VEL
LIN {X 0,Y 194.016,Z 419.338,A -85,B 0,C 180,E1 -21867.07,E2 -21867.07} C_VEL
LIN {X 0,Y 195.091,Z 421.3,A -85,B 0,C 180,E1 -21867.387,E2 -21867.387} C_VEL
LIN {X 0,Y 198.914,Z 433.485,A -85,B 0,C 180,E1 -21869.165,E2 -21869.165} C_VEL
LIN {X 0,Y 201.711,Z 443.239,A -85,B 0,C 180,E1 -21870.802,E2 -21870.802} C_VEL
LIN {X 0,Y 203.732,Z 453.776,A -85,B 0,C 180,E1 -21872.72,E2 -21872.72} C_VEL
LIN {X 0,Y 204.906,Z 462.137,A -85,B 0,C 180,E1 -21874.421,E2 -21874.421} C_VEL
LIN {X 0,Y 202.539,Z 472.574,A -85,B 0,C 180,E1 -21876.476,E2 -21876.476} C_VEL
LIN {X 0,Y 200.049,Z 482.418,A -85,B 0,C 180,E1 -21878.904,E2 -21878.904} C_VEL
LIN {X 0,Y 197.481,Z 491.751,A -85,B 0,C 180,E1 -21881.808,E2 -21881.808} C_VEL
LIN {X 0,Y 195.118,Z 500.045,A -85,B 0,C 180,E1 -21885.138,E2 -21885.138} C_VEL
LIN {X 0,Y 193.61,Z 505.438,A -85,B 0,C 180,E1 -21887.874,E2 -21887.874} C_VEL
LIN {X 0,Y 192.139,Z 510.972,A -85,B 0,C 180,E1 -21891.455,E2 -21891.455} C_VEL
LIN {X 0,Y 191.228,Z 514.956,A -85,B 0,C 180,E1 -21895.002,E2 -21895.002} C_VEL
LIN {X 0,Y 190.525,Z 517.735,A -85,B 0,C 180,E1 -21898.655,E2 -21898.655} C_VEL
LIN {X 0,Y 190.372,Z 519.176,A -85,B 0,C 180,E1 -21901.886,E2 -21901.886} C_VEL
LIN {X 0,Y 190.741,Z 519.662,A -85,B 0,C 180,E1 -21906.124,E2 -21906.124} C_VEL
LIN {X 0,Y 191.566,Z 518.876,A -85,B 0,C 180,E1 -21909.607,E2 -21909.607} C_VEL
LIN {X 0,Y 193.14,Z 516.492,A -85,B 0,C 180,E1 -21913.739,E2 -21913.739} C_VEL
LIN {X 0,Y 195.28,Z 512.656,A -85,B 0,C 180,E1 -21917.673,E2 -21917.673} C_VEL
LIN {X 0,Y 198.062,Z 507.441,A -85,B 0,C 180,E1 -21921.319,E2 -21921.319} C_VEL
LIN {X 0,Y 200.988,Z 501.522,A -85,B 0,C 180,E1 -21924.388,E2 -21924.388} C_VEL
LIN {X 0,Y 204.452,Z 494.011,A -85,B 0,C 180,E1 -21927.393,E2 -21927.393} C_VEL
LIN {X 0,Y 207.97,Z 485.55,A -85,B 0,C 180,E1 -21930.036,E2 -21930.036} C_VEL
LIN {X 0,Y 211.865,Z 475.001,A -85,B 0,C 180,E1 -21932.588,E2 -21932.588} C_VEL
LIN {X 0,Y 212.714,Z 472.4,A -85,B 0,C 180,E1 -21933.133,E2 -21933.133} C_VEL
LIN {X 0,Y 212.019,Z 463.207,A -85,B 0,C 180,E1 -21935.652,E2 -21935.652} C_VEL
LIN {X 0,Y 210.434,Z 454.798,A -85,B 0,C 180,E1 -21937.931,E2 -21937.931} C_VEL
LIN {X 0,Y 207.938,Z 446.562,A -85,B 0,C 180,E1 -21940.246,E2 -21940.246} C_VEL
LIN {X 0,Y 204.056,Z 437.688,A -85,B 0,C 180,E1 -21942.977,E2 -21942.977} C_VEL
LIN {X 0,Y 201.81,Z 433.671,A -85,B 0,C 180,E1 -21944.368,E2 -21944.368} C_VEL
LIN {X 0,Y 199.596,Z 429.878,A -85,B 0,C 180,E1 -21945.731,E2 -21945.731} C_VEL
LIN {X 0,Y 197.577,Z 426.798,A -85,B 0,C 180,E1 -21946.958,E2 -21946.958} C_VEL
LIN {X 0,Y 196.966,Z 425.49,A -85,B 0,C 180,E1 -21947.376,E2 -21947.376} C_VEL
LIN {X 0,Y 194.598,Z 422.927,A -85,B 0,C 180,E1 -21948.706,E2 -21948.706} C_VEL
LIN {X 0,Y 193.595,Z 420.329,A -85,B 0,C 180,E1 -21949.542,E2 -21949.542} C_VEL
LIN {X 0,Y 193.536,Z 419.467,A -85,B 0,C 180,E1 -21953.745,E2 -21953.745} C_VEL
LIN {X 0,Y 193.7,Z 418.808,A -85,B 0,C 180,E1 -21957.92,E2 -21957.92} C_VEL
LIN {X 0,Y 193.835,Z 418.57,A -85,B 0,C 180,E1 -21960,E2 -21960} C_VEL
LIN {X 0,Y 193.373,Z 418.472,A -85,B 0,C 180,E1 -21964.168,E2 -21964.168} C_VEL
LIN {X 0,Y 193.399,Z 418.561,A -85,B 0,C 180,E1 -21968.358,E2 -21968.358} C_VEL
LIN {X 0,Y 193.313,Z 418.971,A -85,B 0,C 180,E1 -21972.599,E2 -21972.599} C_VEL
LIN {X 0,Y 193.364,Z 419.706,A -85,B 0,C 180,E1 -21976.904,E2 -21976.904} C_VEL
LIN {X 0,Y 193.453,Z 420.831,A -85,B 0,C 180,E1 -21981.302,E2 -21981.302} C_VEL
LIN {X 0,Y 193.664,Z 422.318,A -85,B 0,C 180,E1 -21985.816,E2 -21985.816} C_VEL
LIN {X 0,Y 193.944,Z 423.835,A -85,B 0,C 180,E1 -21989.578,E2 -21989.578} C_VEL
LIN {X 0,Y 194.295,Z 425.821,A -85,B 0,C 180,E1 -21993.701,E2 -21993.701} C_VEL
LIN {X 0,Y 194.669,Z 428.147,A -85,B 0,C 180,E1 -21997.86,E2 -21997.86} C_VEL
LIN {X 0,Y 195.213,Z 431.525,A -85,B 0,C 180,E1 -22003.117,E2 -22003.117} C_VEL
LIN {X 0,Y 196.37,Z 434.716,A -85,B 0,C 180,E1 -22003.933,E2 -22003.933} C_VEL
LIN {X 0,Y 198.894,Z 438.297,A -85,B 0,C 180,E1 -22005.331,E2 -22005.331} C_VEL
LIN {X 0,Y 200.822,Z 442.186,A -85,B 0,C 180,E1 -22006.481,E2 -22006.481} C_VEL
LIN {X 0,Y 202.007,Z 444.083,A -85,B 0,C 180,E1 -22007.12,E2 -22007.12} C_VEL
LIN {X 0,Y 204.427,Z 449.874,A -85,B 0,C 180,E1 -22008.674,E2 -22008.674} C_VEL
LIN {X 0,Y 205.927,Z 454.352,A -85,B 0,C 180,E1 -22009.77,E2 -22009.77} C_VEL
LIN {X 0,Y 207.977,Z 465.836,A -85,B 0,C 180,E1 -22012.194,E2 -22012.194} C_VEL
LIN {X 0,Y 208.762,Z 476.986,A -85,B 0,C 180,E1 -22014.551,E2 -22014.551} C_VEL
LIN {X 0,Y 208.501,Z 488.289,A -85,B 0,C 180,E1 -22017.076,E2 -22017.076} C_VEL
LIN {X 0,Y 207.141,Z 497.879,A -85,B 0,C 180,E1 -22019.408,E2 -22019.408} C_VEL
LIN {X 0,Y 205.402,Z 505.167,A -85,B 0,C 180,E1 -22021.379,E2 -22021.379} C_VEL
LIN {X 0,Y 201.567,Z 514.401,A -85,B 0,C 180,E1 -22024.162,E2 -22024.162} C_VEL
LIN {X 0,Y 198.335,Z 522.011,A -85,B 0,C 180,E1 -22027.119,E2 -22027.119} C_VEL
LIN {X 0,Y 195.767,Z 527.969,A -85,B 0,C 180,E1 -22030.059,E2 -22030.059} C_VEL
LIN {X 0,Y 193.605,Z 532.841,A -85,B 0,C 180,E1 -22033.118,E2 -22033.118} C_VEL
LIN {X 0,Y 191.819,Z 537.119,A -85,B 0,C 180,E1 -22036.715,E2 -22036.715} C_VEL
LIN {X 0,Y 191.017,Z 539.455,A -85,B 0,C 180,E1 -22039.399,E2 -22039.399} C_VEL
LIN {X 0,Y 190.413,Z 541.81,A -85,B 0,C 180,E1 -22043.642,E2 -22043.642} C_VEL
LIN {X 0,Y 190.383,Z 542.368,A -85,B 0,C 180,E1 -22045.738,E2 -22045.738} C_VEL
LIN {X 0,Y 189.788,Z 542.501,A -85,B 0,C 180,E1 -22047.508,E2 -22047.508} C_VEL
LIN {X 0,Y 188.251,Z 542.31,A -85,B 0,C 180,E1 -22049.25,E2 -22049.25} C_VEL
LIN {X 0,Y 184.572,Z 541.009,A -85,B 0,C 180,E1 -22052.757,E2 -22052.757} C_VEL
LIN {X 0,Y 183.538,Z 539.9,A -85,B 0,C 180,E1 -22054.571,E2 -22054.571} C_VEL
LIN {X 0,Y 183.457,Z 539.462,A -85,B 0,C 180,E1 -22055.182,E2 -22055.182} C_VEL
LIN {X 0,Y 183.694,Z 536.406,A -85,B 0,C 180,E1 -22058.802,E2 -22058.802} C_VEL
LIN {X 0,Y 184.334,Z 532.488,A -85,B 0,C 180,E1 -22062.104,E2 -22062.104} C_VEL
LIN {X 0,Y 185.488,Z 527.417,A -85,B 0,C 180,E1 -22065.379,E2 -22065.379} C_VEL
LIN {X 0,Y 187.278,Z 521.033,A -85,B 0,C 180,E1 -22068.6,E2 -22068.6} C_VEL
LIN {X 0,Y 189.173,Z 514.522,A -85,B 0,C 180,E1 -22071.236,E2 -22071.236} C_VEL
LIN {X 0,Y 191.363,Z 506.667,A -85,B 0,C 180,E1 -22073.827,E2 -22073.827} C_VEL
LIN {X 0,Y 193.85,Z 497.079,A -85,B 0,C 180,E1 -22076.366,E2 -22076.366} C_VEL
LIN {X 0,Y 194.198,Z 486.371,A -85,B 0,C 180,E1 -22078.861,E2 -22078.861} C_VEL
LIN {X 0,Y 193.941,Z 475.583,A -85,B 0,C 180,E1 -22080.979,E2 -22080.979} C_VEL
LIN {X 0,Y 192.888,Z 462.904,A -85,B 0,C 180,E1 -22083.068,E2 -22083.068} C_VEL
LIN {X 0,Y 190.947,Z 449.386,A -85,B 0,C 180,E1 -22084.937,E2 -22084.937} C_VEL
LIN {X 0,Y 188.111,Z 436.142,A -85,B 0,C 180,E1 -22086.474,E2 -22086.474} C_VEL
LIN {X 0,Y 188.047,Z 435.24,A -85,B 0,C 180,E1 -22086.563,E2 -22086.563} C_VEL
LIN {X 0,Y 188.325,Z 432.596,A -85,B 0,C 180,E1 -22089.375,E2 -22089.375} C_VEL
LIN {X 0,Y 187.911,Z 429.991,A -85,B 0,C 180,E1 -22092.314,E2 -22092.314} C_VEL
LIN {X 0,Y 187.06,Z 425.717,A -85,B 0,C 180,E1 -22097.447,E2 -22097.447} C_VEL
LIN {X 0,Y 186.275,Z 421.515,A -85,B 0,C 180,E1 -22102.867,E2 -22102.867} C_VEL
LIN {X 0,Y 185.718,Z 417.851,A -85,B 0,C 180,E1 -22108.009,E2 -22108.009} C_VEL
LIN {X 0,Y 185.577,Z 417.373,A -85,B 0,C 180,E1 -22108.936,E2 -22108.936} C_VEL
LIN {X 0,Y 185.558,Z 417.373,A -85,B 0,C 180,E1 -22112.967,E2 -22112.967} C_VEL
LIN {X 0,Y 185.595,Z 417.366,A -85,B 0,C 180,E1 -22117.749,E2 -22117.749} C_VEL
LIN {X 0,Y 185.712,Z 417.352,A -85,B 0,C 180,E1 -22122.377,E2 -22122.377} C_VEL
LIN {X 0,Y 185.726,Z 417.351,A -85,B 0,C 180,E1 -22126.877,E2 -22126.877} C_VEL
LIN {X 0,Y 185.978,Z 417.317,A -85,B 0,C 180,E1 -22131.306,E2 -22131.306} C_VEL
LIN {X 0,Y 186.202,Z 417.289,A -85,B 0,C 180,E1 -22137.837,E2 -22137.837} C_VEL
LIN {X 0,Y 186.404,Z 417.264,A -85,B 0,C 180,E1 -22140,E2 -22140} C_VEL
LIN {X 0,Y 185.919,Z 417.314,A -85,B 0,C 180,E1 -22144.336,E2 -22144.336} C_VEL
LIN {X 0,Y 186.004,Z 417.315,A -85,B 0,C 180,E1 -22148.693,E2 -22148.693} C_VEL
LIN {X 0,Y 185.759,Z 417.332,A -85,B 0,C 180,E1 -22153.121,E2 -22153.121} C_VEL
LIN {X 0,Y 185.671,Z 417.356,A -85,B 0,C 180,E1 -22158.868,E2 -22158.868} C_VEL
LIN {X 0,Y 185.598,Z 417.359,A -85,B 0,C 180,E1 -22164.663,E2 -22164.663} C_VEL
LIN {X 0,Y 185.576,Z 417.366,A -85,B 0,C 180,E1 -22169.494,E2 -22169.494} C_VEL
LIN {X 0,Y 185.517,Z 417.373,A -85,B 0,C 180,E1 -22174.629,E2 -22174.629} C_VEL
LIN {X 0,Y 185.541,Z 417.372,A -85,B 0,C 180,E1 -22177.305,E2 -22177.305} C_VEL
LIN {X 0,Y 185.488,Z 417.368,A -85,B 0,C 180,E1 -22180.733,E2 -22180.733} C_VEL
LIN {X 0,Y 185.483,Z 417.382,A -85,B 0,C 180,E1 -22186.048,E2 -22186.048} C_VEL
LIN {X 0,Y 185.466,Z 417.363,A -85,B 0,C 180,E1 -22189.896,E2 -22189.896} C_VEL
LIN {X 0,Y 185.504,Z 417.345,A -85,B 0,C 180,E1 -22192.713,E2 -22192.713} C_VEL
LIN {X 0,Y 185.542,Z 417.376,A -85,B 0,C 180,E1 -22197.976,E2 -22197.976} C_VEL
LIN {X 0,Y 185.581,Z 417.368,A -85,B 0,C 180,E1 -22200.578,E2 -22200.578} C_VEL
LIN {X 0,Y 185.588,Z 417.35,A -85,B 0,C 180,E1 -22205.384,E2 -22205.384} C_VEL
LIN {X 0,Y 185.609,Z 417.363,A -85,B 0,C 180,E1 -22210.077,E2 -22210.077} C_VEL
LIN {X 0,Y 185.727,Z 417.347,A -85,B 0,C 180,E1 -22214.641,E2 -22214.641} C_VEL
LIN {X 0,Y 185.945,Z 417.314,A -85,B 0,C 180,E1 -22219.329,E2 -22219.329} C_VEL
LIN {X 0,Y 186.031,Z 417.314,A -85,B 0,C 180,E1 -22221.309,E2 -22221.309} C_VEL
LIN {X 0,Y 185.848,Z 417.334,A -85,B 0,C 180,E1 -22225.459,E2 -22225.459} C_VEL
LIN {X 0,Y 186.827,Z 420.174,A -85,B 0,C 180,E1 -22225.885,E2 -22225.885} C_VEL
LIN {X 0,Y 189.37,Z 424.997,A -85,B 0,C 180,E1 -22226.744,E2 -22226.744} C_VEL
LIN {X 0,Y 193.078,Z 437.234,A -85,B 0,C 180,E1 -22228.677,E2 -22228.677} C_VEL
LIN {X 0,Y 195.438,Z 446.019,A -85,B 0,C 180,E1 -22230.274,E2 -22230.274} C_VEL
LIN {X 0,Y 197.283,Z 456.39,A -85,B 0,C 180,E1 -22232.297,E2 -22232.297} C_VEL
LIN {X 0,Y 198.146,Z 463.409,A -85,B 0,C 180,E1 -22233.814,E2 -22233.814} C_VEL
LIN {X 0,Y 195.443,Z 474.825,A -85,B 0,C 180,E1 -22236.193,E2 -22236.193} C_VEL
LIN {X 0,Y 192.746,Z 484.833,A -85,B 0,C 180,E1 -22238.85,E2 -22238.85} C_VEL
LIN {X 0,Y 190.276,Z 493.366,A -85,B 0,C 180,E1 -22241.721,E2 -22241.721} C_VEL
LIN {X 0,Y 187.893,Z 501.461,A -85,B 0,C 180,E1 -22245.179,E2 -22245.179} C_VEL
LIN {X 0,Y 186.299,Z 507.152,A -85,B 0,C 180,E1 -22248.312,E2 -22248.312} C_VEL
LIN {X 0,Y 185.125,Z 511.238,A -85,B 0,C 180,E1 -22251.14,E2 -22251.14} C_VEL
LIN {X 0,Y 184.165,Z 515.285,A -85,B 0,C 180,E1 -22254.82,E2 -22254.82} C_VEL
LIN {X 0,Y 183.497,Z 517.904,A -85,B 0,C 180,E1 -22258.247,E2 -22258.247} C_VEL
LIN {X 0,Y 183.29,Z 519.719,A -85,B 0,C 180,E1 -22262.481,E2 -22262.481} C_VEL
LIN {X 0,Y 183.717,Z 520.108,A -85,B 0,C 180,E1 -22266.548,E2 -22266.548} C_VEL
LIN {X 0,Y 184.733,Z 519.212,A -85,B 0,C 180,E1 -22270.457,E2 -22270.457} C_VEL
LIN {X 0,Y 186.232,Z 517.12,A -85,B 0,C 180,E1 -22274.19,E2 -22274.19} C_VEL
LIN {X 0,Y 188.47,Z 513.396,A -85,B 0,C 180,E1 -22278.227,E2 -22278.227} C_VEL
LIN {X 0,Y 191.585,Z 507.956,A -85,B 0,C 180,E1 -22282.205,E2 -22282.205} C_VEL
LIN {X 0,Y 195.289,Z 500.958,A -85,B 0,C 180,E1 -22285.864,E2 -22285.864} C_VEL
LIN {X 0,Y 199.003,Z 493.26,A -85,B 0,C 180,E1 -22288.915,E2 -22288.915} C_VEL
LIN {X 0,Y 202.709,Z 484.655,A -85,B 0,C 180,E1 -22291.559,E2 -22291.559} C_VEL
LIN {X 0,Y 206.651,Z 474.365,A -85,B 0,C 180,E1 -22294.032,E2 -22294.032} C_VEL
LIN {X 0,Y 206.185,Z 465.797,A -85,B 0,C 180,E1 -22296.537,E2 -22296.537} C_VEL
LIN {X 0,Y 204.826,Z 457.776,A -85,B 0,C 180,E1 -22298.883,E2 -22298.883} C_VEL
LIN {X 0,Y 203.123,Z 451.37,A -85,B 0,C 180,E1 -22300.81,E2 -22300.81} C_VEL
LIN {X 0,Y 199.736,Z 442.772,A -85,B 0,C 180,E1 -22303.65,E2 -22303.65} C_VEL
LIN {X 0,Y 195.861,Z 435.475,A -85,B 0,C 180,E1 -22306.421,E2 -22306.421} C_VEL
LIN {X 0,Y 193.772,Z 431.844,A -85,B 0,C 180,E1 -22307.906,E2 -22307.906} C_VEL
LIN {X 0,Y 191.143,Z 428.202,A -85,B 0,C 180,E1 -22309.674,E2 -22309.674} C_VEL
LIN {X 0,Y 190.386,Z 426.515,A -85,B 0,C 180,E1 -22310.304,E2 -22310.304} C_VEL
LIN {X 0,Y 187.833,Z 423.941,A -85,B 0,C 180,E1 -22312.002,E2 -22312.002} C_VEL
LIN {X 0,Y 186.702,Z 421.466,A -85,B 0,C 180,E1 -22312.973,E2 -22312.973} C_VEL
LIN {X 0,Y 186.633,Z 421.146,A -85,B 0,C 180,E1 -22313.513,E2 -22313.513} C_VEL
LIN {X 0,Y 186.795,Z 420.508,A -85,B 0,C 180,E1 -22317.844,E2 -22317.844} C_VEL
LIN {X 0,Y 186.95,Z 420.278,A -85,B 0,C 180,E1 -22320,E2 -22320} C_VEL
LIN {X 0,Y 186.499,Z 420.211,A -85,B 0,C 180,E1 -22324.322,E2 -22324.322} C_VEL
LIN {X 0,Y 186.519,Z 420.333,A -85,B 0,C 180,E1 -22328.668,E2 -22328.668} C_VEL
LIN {X 0,Y 186.446,Z 420.807,A -85,B 0,C 180,E1 -22333.071,E2 -22333.071} C_VEL
LIN {X 0,Y 186.486,Z 421.616,A -85,B 0,C 180,E1 -22337.547,E2 -22337.547} C_VEL
LIN {X 0,Y 186.588,Z 422.809,A -85,B 0,C 180,E1 -22342.127,E2 -22342.127} C_VEL
LIN {X 0,Y 186.838,Z 424.401,A -85,B 0,C 180,E1 -22346.833,E2 -22346.833} C_VEL
LIN {X 0,Y 187.093,Z 425.802,A -85,B 0,C 180,E1 -22350.235,E2 -22350.235} C_VEL
LIN {X 0,Y 187.406,Z 427.802,A -85,B 0,C 180,E1 -22354.409,E2 -22354.409} C_VEL
LIN {X 0,Y 187.839,Z 430.588,A -85,B 0,C 180,E1 -22359.397,E2 -22359.397} C_VEL
LIN {X 0,Y 189.335,Z 434.322,A -85,B 0,C 180,E1 -22360.691,E2 -22360.691} C_VEL
LIN {X 0,Y 191.858,Z 437.659,A -85,B 0,C 180,E1 -22362.308,E2 -22362.308} C_VEL
LIN {X 0,Y 193.737,Z 441.674,A -85,B 0,C 180,E1 -22363.657,E2 -22363.657} C_VEL
LIN {X 0,Y 195.234,Z 444.005,A -85,B 0,C 180,E1 -22364.587,E2 -22364.587} C_VEL
LIN {X 0,Y 197.388,Z 448.305,A -85,B 0,C 180,E1 -22366.045,E2 -22366.045} C_VEL
LIN {X 0,Y 200.298,Z 455.663,A -85,B 0,C 180,E1 -22368.19,E2 -22368.19} C_VEL
LIN {X 0,Y 201.633,Z 461.953,A -85,B 0,C 180,E1 -22369.7,E2 -22369.7} C_VEL
LIN {X 0,Y 202.697,Z 471.608,A -85,B 0,C 180,E1 -22371.878,E2 -22371.878} C_VEL
LIN {X 0,Y 202.87,Z 481.84,A -85,B 0,C 180,E1 -22374.226,E2 -22374.226} C_VEL
LIN {X 0,Y 202.027,Z 492.526,A -85,B 0,C 180,E1 -22376.831,E2 -22376.831} C_VEL
LIN {X 0,Y 200.159,Z 502.088,A -85,B 0,C 180,E1 -22379.395,E2 -22379.395} C_VEL
LIN {X 0,Y 198.57,Z 507.169,A -85,B 0,C 180,E1 -22380.879,E2 -22380.879} C_VEL
LIN {X 0,Y 194.592,Z 515.939,A -85,B 0,C 180,E1 -22383.741,E2 -22383.741} C_VEL
LIN {X 0,Y 191.576,Z 522.545,A -85,B 0,C 180,E1 -22386.51,E2 -22386.51} C_VEL
LIN {X 0,Y 189.091,Z 527.917,A -85,B 0,C 180,E1 -22389.324,E2 -22389.324} C_VEL
LIN {X 0,Y 186.797,Z 532.708,A -85,B 0,C 180,E1 -22392.483,E2 -22392.483} C_VEL
LIN {X 0,Y 185.072,Z 536.425,A -85,B 0,C 180,E1 -22395.71,E2 -22395.71} C_VEL
LIN {X 0,Y 184.024,Z 539.172,A -85,B 0,C 180,E1 -22398.991,E2 -22398.991} C_VEL
LIN {X 0,Y 183.356,Z 541.441,A -85,B 0,C 180,E1 -22403.397,E2 -22403.397} C_VEL
LIN {X 0,Y 183.306,Z 541.96,A -85,B 0,C 180,E1 -22405.734,E2 -22405.734} C_VEL
LIN {X 0,Y 183.407,Z 542.078,A -85,B 0,C 180,E1 -22407.803,E2 -22407.803} C_VEL
LIN {X 0,Y 183.547,Z 541.812,A -85,B 0,C 180,E1 -22409.999,E2 -22409.999} C_VEL
LIN {X 0,Y 183.468,Z 541.126,A -85,B 0,C 180,E1 -22412.195,E2 -22412.195} C_VEL
LIN {X 0,Y 183.457,Z 539.462,A -85,B 0,C 180,E1 -22415.182,E2 -22415.182} C_VEL
LIN {X 0,Y 182.848,Z 538.085,A -85,B 0,C 180,E1 -22416.962,E2 -22416.962} C_VEL
LIN {X 0,Y 180.317,Z 535.147,A -85,B 0,C 180,E1 -22419.845,E2 -22419.845} C_VEL
LIN {X 0,Y 178.383,Z 532.318,A -85,B 0,C 180,E1 -22422.153,E2 -22422.153} C_VEL
LIN {X 0,Y 177.857,Z 529.897,A -85,B 0,C 180,E1 -22423.894,E2 -22423.894} C_VEL
LIN {X 0,Y 177.973,Z 529.01,A -85,B 0,C 180,E1 -22424.469,E2 -22424.469} C_VEL
LIN {X 0,Y 179.572,Z 523.521,A -85,B 0,C 180,E1 -22427.656,E2 -22427.656} C_VEL
LIN {X 0,Y 181.772,Z 516.255,A -85,B 0,C 180,E1 -22430.954,E2 -22430.954} C_VEL
LIN {X 0,Y 184.268,Z 507.367,A -85,B 0,C 180,E1 -22434.144,E2 -22434.144} C_VEL
LIN {X 0,Y 186.938,Z 497.88,A -85,B 0,C 180,E1 -22436.816,E2 -22436.816} C_VEL
LIN {X 0,Y 187.403,Z 488.35,A -85,B 0,C 180,E1 -22439.177,E2 -22439.177} C_VEL
LIN {X 0,Y 187.291,Z 477.468,A -85,B 0,C 180,E1 -22441.475,E2 -22441.475} C_VEL
LIN {X 0,Y 186.437,Z 464.797,A -85,B 0,C 180,E1 -22443.742,E2 -22443.742} C_VEL
LIN {X 0,Y 184.715,Z 451.658,A -85,B 0,C 180,E1 -22445.707,E2 -22445.707} C_VEL
LIN {X 0,Y 182.071,Z 438.528,A -85,B 0,C 180,E1 -22447.364,E2 -22447.364} C_VEL
LIN {X 0,Y 181.183,Z 434.745,A -85,B 0,C 180,E1 -22447.848,E2 -22447.848} C_VEL
LIN {X 0,Y 181.277,Z 433.564,A -85,B 0,C 180,E1 -22449.16,E2 -22449.16} C_VEL
LIN {X 0,Y 180.843,Z 430.83,A -85,B 0,C 180,E1 -22452.406,E2 -22452.406} C_VEL
LIN {X 0,Y 180.357,Z 428.341,A -85,B 0,C 180,E1 -22455.46,E2 -22455.46} C_VEL
LIN {X 0,Y 179.657,Z 424.991,A -85,B 0,C 180,E1 -22459.8,E2 -22459.8} C_VEL
LIN {X 0,Y 178.963,Z 420.851,A -85,B 0,C 180,E1 -22465.554,E2 -22465.554} C_VEL
LIN {X 0,Y 178.536,Z 418.249,A -85,B 0,C 180,E1 -22469.719,E2 -22469.719} C_VEL
LIN {X 0,Y 178.531,Z 418.247,A -85,B 0,C 180,E1 -22474.875,E2 -22474.875} C_VEL
LIN {X 0,Y 178.634,Z 418.235,A -85,B 0,C 180,E1 -22480.77,E2 -22480.77} C_VEL
LIN {X 0,Y 178.655,Z 418.231,A -85,B 0,C 180,E1 -22486.348,E2 -22486.348} C_VEL
LIN {X 0,Y 178.907,Z 418.199,A -85,B 0,C 180,E1 -22490.96,E2 -22490.96} C_VEL
LIN {X 0,Y 179.147,Z 418.168,A -85,B 0,C 180,E1 -22497.752,E2 -22497.752} C_VEL
LIN {X 0,Y 179.367,Z 418.141,A -85,B 0,C 180,E1 -22500,E2 -22500} C_VEL
LIN {X 0,Y 178.867,Z 418.193,A -85,B 0,C 180,E1 -22504.507,E2 -22504.507} C_VEL
LIN {X 0,Y 178.955,Z 418.192,A -85,B 0,C 180,E1 -22509.038,E2 -22509.038} C_VEL
LIN {X 0,Y 178.676,Z 418.214,A -85,B 0,C 180,E1 -22513.651,E2 -22513.651} C_VEL
LIN {X 0,Y 178.619,Z 418.233,A -85,B 0,C 180,E1 -22519.217,E2 -22519.217} C_VEL
LIN {X 0,Y 178.531,Z 418.241,A -85,B 0,C 180,E1 -22525.125,E2 -22525.125} C_VEL
LIN {X 0,Y 178.52,Z 418.244,A -85,B 0,C 180,E1 -22529.995,E2 -22529.995} C_VEL
LIN {X 0,Y 178.493,Z 418.244,A -85,B 0,C 180,E1 -22534.226,E2 -22534.226} C_VEL
LIN {X 0,Y 178.418,Z 418.256,A -85,B 0,C 180,E1 -22539.069,E2 -22539.069} C_VEL
LIN {X 0,Y 178.415,Z 418.251,A -85,B 0,C 180,E1 -22542.041,E2 -22542.041} C_VEL
LIN {X 0,Y 178.411,Z 418.261,A -85,B 0,C 180,E1 -22545.159,E2 -22545.159} C_VEL
LIN {X 0,Y 178.407,Z 418.252,A -85,B 0,C 180,E1 -22548.459,E2 -22548.459} C_VEL
LIN {X 0,Y 178.421,Z 418.233,A -85,B 0,C 180,E1 -22553.784,E2 -22553.784} C_VEL
LIN {X 0,Y 178.485,Z 418.249,A -85,B 0,C 180,E1 -22556.548,E2 -22556.548} C_VEL
LIN {X 0,Y 178.522,Z 418.25,A -85,B 0,C 180,E1 -22560.008,E2 -22560.008} C_VEL
LIN {X 0,Y 178.535,Z 418.225,A -85,B 0,C 180,E1 -22564.877,E2 -22564.877} C_VEL
LIN {X 0,Y 178.625,Z 418.23,A -85,B 0,C 180,E1 -22570.785,E2 -22570.785} C_VEL
LIN {X 0,Y 178.668,Z 418.219,A -85,B 0,C 180,E1 -22574.018,E2 -22574.018} C_VEL
LIN {X 0,Y 178.897,Z 418.191,A -85,B 0,C 180,E1 -22579.154,E2 -22579.154} C_VEL
LIN {X 0,Y 178.919,Z 418.194,A -85,B 0,C 180,E1 -22583.233,E2 -22583.233} C_VEL
LIN {X 0,Y 178.865,Z 418.226,A -85,B 0,C 180,E1 -22584.222,E2 -22584.222} C_VEL
LIN {X 0,Y 179.89,Z 421.148,A -85,B 0,C 180,E1 -22584.653,E2 -22584.653} C_VEL
LIN {X 0,Y 183.799,Z 429.211,A -85,B 0,C 180,E1 -22586.161,E2 -22586.161} C_VEL
LIN {X 0,Y 187.479,Z 441.877,A -85,B 0,C 180,E1 -22588.392,E2 -22588.392} C_VEL
LIN {X 0,Y 189.409,Z 450.13,A -85,B 0,C 180,E1 -22590.001,E2 -22590.001} C_VEL
LIN {X 0,Y 190.974,Z 460.09,A -85,B 0,C 180,E1 -22592.109,E2 -22592.109} C_VEL
LIN {X 0,Y 191.498,Z 464.074,A -85,B 0,C 180,E1 -22593.039,E2 -22593.039} C_VEL
LIN {X 0,Y 188.968,Z 474.743,A -85,B 0,C 180,E1 -22595.335,E2 -22595.335} C_VEL
LIN {X 0,Y 186.621,Z 483.18,A -85,B 0,C 180,E1 -22597.574,E2 -22597.574} C_VEL
LIN {X 0,Y 183.943,Z 492.152,A -85,B 0,C 180,E1 -22600.524,E2 -22600.524} C_VEL
LIN {X 0,Y 181.8,Z 499.135,A -85,B 0,C 180,E1 -22603.412,E2 -22603.412} C_VEL
LIN {X 0,Y 179.715,Z 506.048,A -85,B 0,C 180,E1 -22607.056,E2 -22607.056} C_VEL
LIN {X 0,Y 178.111,Z 511.497,A -85,B 0,C 180,E1 -22610.801,E2 -22610.801} C_VEL
LIN {X 0,Y 177.211,Z 515.184,A -85,B 0,C 180,E1 -22614.194,E2 -22614.194} C_VEL
LIN {X 0,Y 176.35,Z 518.561,A -85,B 0,C 180,E1 -22618.745,E2 -22618.745} C_VEL
LIN {X 0,Y 176.244,Z 520.257,A -85,B 0,C 180,E1 -22623.132,E2 -22623.132} C_VEL
LIN {X 0,Y 176.788,Z 520.542,A -85,B 0,C 180,E1 -22627.337,E2 -22627.337} C_VEL
LIN {X 0,Y 177.923,Z 519.523,A -85,B 0,C 180,E1 -22631.365,E2 -22631.365} C_VEL
LIN {X 0,Y 179.577,Z 517.35,A -85,B 0,C 180,E1 -22635.214,E2 -22635.214} C_VEL
LIN {X 0,Y 181.72,Z 514.07,A -85,B 0,C 180,E1 -22638.892,E2 -22638.892} C_VEL
LIN {X 0,Y 184.574,Z 509.53,A -85,B 0,C 180,E1 -22642.466,E2 -22642.466} C_VEL
LIN {X 0,Y 187.902,Z 503.72,A -85,B 0,C 180,E1 -22645.872,E2 -22645.872} C_VEL
LIN {X 0,Y 191.799,Z 496.301,A -85,B 0,C 180,E1 -22649.136,E2 -22649.136} C_VEL
LIN {X 0,Y 195.361,Z 488.89,A -85,B 0,C 180,E1 -22651.682,E2 -22651.682} C_VEL
LIN {X 0,Y 199.187,Z 479.977,A -85,B 0,C 180,E1 -22654.121,E2 -22654.121} C_VEL
LIN {X 0,Y 200.618,Z 475.808,A -85,B 0,C 180,E1 -22655.141,E2 -22655.141} C_VEL
LIN {X 0,Y 200.279,Z 467.668,A -85,B 0,C 180,E1 -22657.702,E2 -22657.702} C_VEL
LIN {X 0,Y 199.094,Z 459.922,A -85,B 0,C 180,E1 -22660.137,E2 -22660.137} C_VEL
LIN {X 0,Y 197.235,Z 452.918,A -85,B 0,C 180,E1 -22662.471,E2 -22662.471} C_VEL
LIN {X 0,Y 194.134,Z 445.238,A -85,B 0,C 180,E1 -22665.32,E2 -22665.32} C_VEL
LIN {X 0,Y 189.553,Z 436.701,A -85,B 0,C 180,E1 -22669.046,E2 -22669.046} C_VEL
LIN {X 0,Y 187.614,Z 433.481,A -85,B 0,C 180,E1 -22670.635,E2 -22670.635} C_VEL
LIN {X 0,Y 186.922,Z 432.333,A -85,B 0,C 180,E1 -22671.214,E2 -22671.214} C_VEL
LIN {X 0,Y 184.554,Z 429.284,A -85,B 0,C 180,E1 -22673.096,E2 -22673.096} C_VEL
LIN {X 0,Y 183.769,Z 427.588,A -85,B 0,C 180,E1 -22673.893,E2 -22673.893} C_VEL
LIN {X 0,Y 181.371,Z 425.554,A -85,B 0,C 180,E1 -22675.833,E2 -22675.833} C_VEL
LIN {X 0,Y 180.042,Z 422.966,A -85,B 0,C 180,E1 -22677.273,E2 -22677.273} C_VEL
LIN {X 0,Y 179.863,Z 422.23,A -85,B 0,C 180,E1 -22677.62,E2 -22677.62} C_VEL
LIN {X 0,Y 180.051,Z 421.986,A -85,B 0,C 180,E1 -22680,E2 -22680} C_VEL
LIN {X 0,Y 179.61,Z 421.955,A -85,B 0,C 180,E1 -22684.488,E2 -22684.488} C_VEL
LIN {X 0,Y 179.628,Z 422.124,A -85,B 0,C 180,E1 -22689.004,E2 -22689.004} C_VEL
LIN {X 0,Y 179.556,Z 422.65,A -85,B 0,C 180,E1 -22693.582,E2 -22693.582} C_VEL
LIN {X 0,Y 179.591,Z 423.537,A -85,B 0,C 180,E1 -22698.244,E2 -22698.244} C_VEL
LIN {X 0,Y 179.739,Z 424.814,A -85,B 0,C 180,E1 -22703.017,E2 -22703.017} C_VEL
LIN {X 0,Y 179.909,Z 425.825,A -85,B 0,C 180,E1 -22706.043,E2 -22706.043} C_VEL
LIN {X 0,Y 180.195,Z 427.755,A -85,B 0,C 180,E1 -22710.903,E2 -22710.903} C_VEL
LIN {X 0,Y 180.559,Z 429.81,A -85,B 0,C 180,E1 -22714.867,E2 -22714.867} C_VEL
LIN {X 0,Y 181.682,Z 432.708,A -85,B 0,C 180,E1 -22716.065,E2 -22716.065} C_VEL
LIN {X 0,Y 184.576,Z 436.454,A -85,B 0,C 180,E1 -22718.423,E2 -22718.423} C_VEL
LIN {X 0,Y 187.005,Z 441.417,A -85,B 0,C 180,E1 -22720.502,E2 -22720.502} C_VEL
LIN {X 0,Y 188.421,Z 443.448,A -85,B 0,C 180,E1 -22721.523,E2 -22721.523} C_VEL
LIN {X 0,Y 190.321,Z 447.612,A -85,B 0,C 180,E1 -22723.081,E2 -22723.081} C_VEL
LIN {X 0,Y 193.097,Z 453.275,A -85,B 0,C 180,E1 -22725.212,E2 -22725.212} C_VEL
LIN {X 0,Y 195.606,Z 460.351,A -85,B 0,C 180,E1 -22727.437,E2 -22727.437} C_VEL
LIN {X 0,Y 196.719,Z 468.034,A -85,B 0,C 180,E1 -22729.369,E2 -22729.369} C_VEL
LIN {X 0,Y 197.168,Z 479.132,A -85,B 0,C 180,E1 -22732.079,E2 -22732.079} C_VEL
LIN {X 0,Y 196.479,Z 489.812,A -85,B 0,C 180,E1 -22734.775,E2 -22734.775} C_VEL
LIN {X 0,Y 194.916,Z 498.905,A -85,B 0,C 180,E1 -22737.259,E2 -22737.259} C_VEL
LIN {X 0,Y 193.015,Z 505.901,A -85,B 0,C 180,E1 -22739.352,E2 -22739.352} C_VEL
LIN {X 0,Y 188.879,Z 514.798,A -85,B 0,C 180,E1 -22742.283,E2 -22742.283} C_VEL
LIN {X 0,Y 185.355,Z 522.038,A -85,B 0,C 180,E1 -22745.35,E2 -22745.35} C_VEL
LIN {X 0,Y 182.455,Z 527.905,A -85,B 0,C 180,E1 -22748.535,E2 -22748.535} C_VEL
LIN {X 0,Y 180.018,Z 532.59,A -85,B 0,C 180,E1 -22751.8,E2 -22751.8} C_VEL
LIN {X 0,Y 178.15,Z 536.215,A -85,B 0,C 180,E1 -22755.142,E2 -22755.142} C_VEL
LIN {X 0,Y 177.017,Z 538.889,A -85,B 0,C 180,E1 -22758.55,E2 -22758.55} C_VEL
LIN {X 0,Y 176.541,Z 540.187,A -85,B 0,C 180,E1 -22760.837,E2 -22760.837} C_VEL
LIN {X 0,Y 176.297,Z 541.056,A -85,B 0,C 180,E1 -22763.131,E2 -22763.131} C_VEL
LIN {X 0,Y 176.322,Z 541.624,A -85,B 0,C 180,E1 -22767.715,E2 -22767.715} C_VEL
LIN {X 0,Y 176.481,Z 541.326,A -85,B 0,C 180,E1 -22769.999,E2 -22769.999} C_VEL
LIN {X 0,Y 176.385,Z 540.58,A -85,B 0,C 180,E1 -22772.283,E2 -22772.283} C_VEL
LIN {X 0,Y 176.393,Z 539.037,A -85,B 0,C 180,E1 -22775.131,E2 -22775.131} C_VEL
LIN {X 0,Y 176.663,Z 535.743,A -85,B 0,C 180,E1 -22779.155,E2 -22779.155} C_VEL
LIN {X 0,Y 177.374,Z 531.749,A -85,B 0,C 180,E1 -22782.586,E2 -22782.586} C_VEL
LIN {X 0,Y 177.973,Z 529.01,A -85,B 0,C 180,E1 -22784.469,E2 -22784.469} C_VEL
LIN {X 0,Y 178,Z 526.3,A -85,B 0,C 180,E1 -22786.162,E2 -22786.162} C_VEL
LIN {X 0,Y 176.584,Z 521.338,A -85,B 0,C 180,E1 -22788.903,E2 -22788.903} C_VEL
LIN {X 0,Y 175.463,Z 515.743,A -85,B 0,C 180,E1 -22791.553,E2 -22791.553} C_VEL
LIN {X 0,Y 175.945,Z 512.037,A -85,B 0,C 180,E1 -22793.053,E2 -22793.053} C_VEL
LIN {X 0,Y 178.884,Z 502.463,A -85,B 0,C 180,E1 -22796.23,E2 -22796.23} C_VEL
LIN {X 0,Y 180.194,Z 497.549,A -85,B 0,C 180,E1 -22797.59,E2 -22797.59} C_VEL
LIN {X 0,Y 180.677,Z 486.652,A -85,B 0,C 180,E1 -22800.375,E2 -22800.375} C_VEL
LIN {X 0,Y 180.497,Z 475.753,A -85,B 0,C 180,E1 -22802.742,E2 -22802.742} C_VEL
LIN {X 0,Y 179.677,Z 463.238,A -85,B 0,C 180,E1 -22805.019,E2 -22805.019} C_VEL
LIN {X 0,Y 177.849,Z 450.133,A -85,B 0,C 180,E1 -22807.042,E2 -22807.042} C_VEL
LIN {X 0,Y 175.561,Z 439.399,A -85,B 0,C 180,E1 -22808.506,E2 -22808.506} C_VEL
LIN {X 0,Y 174.223,Z 434.363,A -85,B 0,C 180,E1 -22809.169,E2 -22809.169} C_VEL
LIN {X 0,Y 173.601,Z 430.88,A -85,B 0,C 180,E1 -22813.488,E2 -22813.488} C_VEL
LIN {X 0,Y 173.074,Z 428.187,A -85,B 0,C 180,E1 -22816.962,E2 -22816.962} C_VEL
LIN {X 0,Y 172.305,Z 424.344,A -85,B 0,C 180,E1 -22822.279,E2 -22822.279} C_VEL
LIN {X 0,Y 172.008,Z 422.416,A -85,B 0,C 180,E1 -22825.109,E2 -22825.109} C_VEL
LIN {X 0,Y 171.487,Z 419.128,A -85,B 0,C 180,E1 -22830.233,E2 -22830.233} C_VEL
LIN {X 0,Y 171.455,Z 419.127,A -85,B 0,C 180,E1 -22835.801,E2 -22835.801} C_VEL
LIN {X 0,Y 171.591,Z 419.112,A -85,B 0,C 180,E1 -22840.873,E2 -22840.873} C_VEL
LIN {X 0,Y 171.575,Z 419.112,A -85,B 0,C 180,E1 -22845.773,E2 -22845.773} C_VEL
LIN {X 0,Y 171.843,Z 419.081,A -85,B 0,C 180,E1 -22850.585,E2 -22850.585} C_VEL
LIN {X 0,Y 171.81,Z 419.074,A -85,B 0,C 180,E1 -22855.308,E2 -22855.308} C_VEL
LIN {X 0,Y 172.33,Z 419.018,A -85,B 0,C 180,E1 -22860,E2 -22860} C_VEL
LIN {X 0,Y 171.816,Z 419.072,A -85,B 0,C 180,E1 -22864.693,E2 -22864.693} C_VEL
LIN {X 0,Y 171.884,Z 419.072,A -85,B 0,C 180,E1 -22869.413,E2 -22869.413} C_VEL
LIN {X 0,Y 171.589,Z 419.098,A -85,B 0,C 180,E1 -22874.227,E2 -22874.227} C_VEL
LIN {X 0,Y 171.541,Z 419.115,A -85,B 0,C 180,E1 -22879.563,E2 -22879.563} C_VEL
LIN {X 0,Y 171.466,Z 419.122,A -85,B 0,C 180,E1 -22885.617,E2 -22885.617} C_VEL
LIN {X 0,Y 171.439,Z 419.122,A -85,B 0,C 180,E1 -22890.588,E2 -22890.588} C_VEL
LIN {X 0,Y 171.404,Z 419.131,A -85,B 0,C 180,E1 -22895.033,E2 -22895.033} C_VEL
LIN {X 0,Y 171.379,Z 419.133,A -85,B 0,C 180,E1 -22898.819,E2 -22898.819} C_VEL
LIN {X 0,Y 171.336,Z 419.143,A -85,B 0,C 180,E1 -22904.213,E2 -22904.213} C_VEL
LIN {X 0,Y 171.337,Z 419.131,A -85,B 0,C 180,E1 -22908.984,E2 -22908.984} C_VEL
LIN {X 0,Y 171.385,Z 419.101,A -85,B 0,C 180,E1 -22912.042,E2 -22912.042} C_VEL
LIN {X 0,Y 171.397,Z 419.119,A -85,B 0,C 180,E1 -22915.094,E2 -22915.094} C_VEL
LIN {X 0,Y 171.448,Z 419.129,A -85,B 0,C 180,E1 -22920.536,E2 -22920.536} C_VEL
LIN {X 0,Y 171.459,Z 419.111,A -85,B 0,C 180,E1 -22925.803,E2 -22925.803} C_VEL
LIN {X 0,Y 171.581,Z 419.107,A -85,B 0,C 180,E1 -22930.873,E2 -22930.873} C_VEL
LIN {X 0,Y 171.613,Z 419.11,A -85,B 0,C 180,E1 -22935.777,E2 -22935.777} C_VEL
LIN {X 0,Y 171.913,Z 419.068,A -85,B 0,C 180,E1 -22940.589,E2 -22940.589} C_VEL
LIN {X 0,Y 171.88,Z 419.074,A -85,B 0,C 180,E1 -22942.807,E2 -22942.807} C_VEL
LIN {X 0,Y 172.955,Z 422.037,A -85,B 0,C 180,E1 -22943.336,E2 -22943.336} C_VEL
LIN {X 0,Y 178.021,Z 432.757,A -85,B 0,C 180,E1 -22945.472,E2 -22945.472} C_VEL
LIN {X 0,Y 181.358,Z 444.824,A -85,B 0,C 180,E1 -22947.78,E2 -22947.78} C_VEL
LIN {X 0,Y 183.366,Z 454.224,A -85,B 0,C 180,E1 -22949.763,E2 -22949.763} C_VEL
LIN {X 0,Y 184.726,Z 464.639,A -85,B 0,C 180,E1 -22952.181,E2 -22952.181} C_VEL
LIN {X 0,Y 184.179,Z 468.145,A -85,B 0,C 180,E1 -22952.934,E2 -22952.934} C_VEL
LIN {X 0,Y 181.525,Z 478.005,A -85,B 0,C 180,E1 -22955.276,E2 -22955.276} C_VEL
LIN {X 0,Y 178.914,Z 486.871,A -85,B 0,C 180,E1 -22957.903,E2 -22957.903} C_VEL
LIN {X 0,Y 176.346,Z 495.029,A -85,B 0,C 180,E1 -22960.913,E2 -22960.913} C_VEL
LIN {X 0,Y 174.036,Z 502.242,A -85,B 0,C 180,E1 -22964.26,E2 -22964.26} C_VEL
LIN {X 0,Y 172.218,Z 508.217,A -85,B 0,C 180,E1 -22967.822,E2 -22967.822} C_VEL
LIN {X 0,Y 170.728,Z 513.239,A -85,B 0,C 180,E1 -22971.746,E2 -22971.746} C_VEL
LIN {X 0,Y 169.99,Z 516.017,A -85,B 0,C 180,E1 -22974.555,E2 -22974.555} C_VEL
LIN {X 0,Y 169.194,Z 519.206,A -85,B 0,C 180,E1 -22979.272,E2 -22979.272} C_VEL
LIN {X 0,Y 169.205,Z 520.795,A -85,B 0,C 180,E1 -22983.827,E2 -22983.827} C_VEL
LIN {X 0,Y 169.9,Z 520.915,A -85,B 0,C 180,E1 -22988.351,E2 -22988.351} C_VEL
LIN {X 0,Y 171.167,Z 519.834,A -85,B 0,C 180,E1 -22992.347,E2 -22992.347} C_VEL
LIN {X 0,Y 173.326,Z 517.194,A -85,B 0,C 180,E1 -22996.874,E2 -22996.874} C_VEL
LIN {X 0,Y 176.203,Z 513.03,A -85,B 0,C 180,E1 -23001.201,E2 -23001.201} C_VEL
LIN {X 0,Y 179.792,Z 507.463,A -85,B 0,C 180,E1 -23005.172,E2 -23005.172} C_VEL
LIN {X 0,Y 183.471,Z 501.259,A -85,B 0,C 180,E1 -23008.462,E2 -23008.462} C_VEL
LIN {X 0,Y 187.741,Z 493.357,A -85,B 0,C 180,E1 -23011.644,E2 -23011.644} C_VEL
LIN {X 0,Y 191.985,Z 484.456,A -85,B 0,C 180,E1 -23014.429,E2 -23014.429} C_VEL
LIN {X 0,Y 194.659,Z 478.19,A -85,B 0,C 180,E1 -23016.024,E2 -23016.024} C_VEL
LIN {X 0,Y 194.623,Z 471.507,A -85,B 0,C 180,E1 -23018.276,E2 -23018.276} C_VEL
LIN {X 0,Y 193.735,Z 463.658,A -85,B 0,C 180,E1 -23020.944,E2 -23020.944} C_VEL
LIN {X 0,Y 192.017,Z 456.52,A -85,B 0,C 180,E1 -23023.521,E2 -23023.521} C_VEL
LIN {X 0,Y 189.512,Z 449.742,A -85,B 0,C 180,E1 -23026.267,E2 -23026.267} C_VEL
LIN {X 0,Y 186.531,Z 443.541,A -85,B 0,C 180,E1 -23029.141,E2 -23029.141} C_VEL
LIN {X 0,Y 183.061,Z 437.665,A -85,B 0,C 180,E1 -23032.347,E2 -23032.347} C_VEL
LIN {X 0,Y 181.121,Z 434.21,A -85,B 0,C 180,E1 -23034.354,E2 -23034.354} C_VEL
LIN {X 0,Y 178.389,Z 431.197,A -85,B 0,C 180,E1 -23036.965,E2 -23036.965} C_VEL
LIN {X 0,Y 177.452,Z 428.818,A -85,B 0,C 180,E1 -23038.298,E2 -23038.298} C_VEL
LIN {X 0,Y 173.562,Z 425.422,A -85,B 0,C 180,E1 -23043.046,E2 -23043.046} C_VEL
LIN {X 0,Y 172.719,Z 423.698,A -85,B 0,C 180,E1 -23044.668,E2 -23044.668} C_VEL
LIN {X 0,Y 172.729,Z 423.92,A -85,B 0,C 180,E1 -23049.366,E2 -23049.366} C_VEL
LIN {X 0,Y 172.664,Z 424.513,A -85,B 0,C 180,E1 -23054.136,E2 -23054.136} C_VEL
LIN {X 0,Y 172.72,Z 425.472,A -85,B 0,C 180,E1 -23058.997,E2 -23058.997} C_VEL
LIN {X 0,Y 172.895,Z 426.837,A -85,B 0,C 180,E1 -23063.984,E2 -23063.984} C_VEL
LIN {X 0,Y 173.092,Z 428.215,A -85,B 0,C 180,E1 -23067.743,E2 -23067.743} C_VEL
LIN {X 0,Y 174.373,Z 431.496,A -85,B 0,C 180,E1 -23069.918,E2 -23069.918} C_VEL
LIN {X 0,Y 177.031,Z 435.06,A -85,B 0,C 180,E1 -23073.084,E2 -23073.084} C_VEL
LIN {X 0,Y 177.954,Z 436.099,A -85,B 0,C 180,E1 -23073.999,E2 -23073.999} C_VEL
LIN {X 0,Y 179.511,Z 439.764,A -85,B 0,C 180,E1 -23075.836,E2 -23075.836} C_VEL
LIN {X 0,Y 181.735,Z 442.957,A -85,B 0,C 180,E1 -23077.873,E2 -23077.873} C_VEL
LIN {X 0,Y 183.711,Z 447.286,A -85,B 0,C 180,E1 -23079.824,E2 -23079.824} C_VEL
LIN {X 0,Y 184.418,Z 448.264,A -85,B 0,C 180,E1 -23080.38,E2 -23080.38} C_VEL
LIN {X 0,Y 188.623,Z 457.992,A -85,B 0,C 180,E1 -23084.316,E2 -23084.316} C_VEL
LIN {X 0,Y 190.645,Z 464.324,A -85,B 0,C 180,E1 -23086.493,E2 -23086.493} C_VEL
LIN {X 0,Y 191.461,Z 472.327,A -85,B 0,C 180,E1 -23088.645,E2 -23088.645} C_VEL
LIN {X 0,Y 191.393,Z 482.711,A -85,B 0,C 180,E1 -23091.374,E2 -23091.374} C_VEL
LIN {X 0,Y 190.14,Z 493.761,A -85,B 0,C 180,E1 -23094.407,E2 -23094.407} C_VEL
LIN {X 0,Y 188.441,Z 501.298,A -85,B 0,C 180,E1 -23096.626,E2 -23096.626} C_VEL
LIN {X 0,Y 186.289,Z 507.915,A -85,B 0,C 180,E1 -23098.753,E2 -23098.753} C_VEL
LIN {X 0,Y 181.973,Z 516.308,A -85,B 0,C 180,E1 -23101.764,E2 -23101.764} C_VEL
LIN {X 0,Y 178.136,Z 523.544,A -85,B 0,C 180,E1 -23105.151,E2 -23105.151} C_VEL
LIN {X 0,Y 174.885,Z 529.516,A -85,B 0,C 180,E1 -23108.797,E2 -23108.797} C_VEL
LIN {X 0,Y 172.537,Z 533.75,A -85,B 0,C 180,E1 -23112.212,E2 -23112.212} C_VEL
LIN {X 0,Y 170.778,Z 536.971,A -85,B 0,C 180,E1 -23115.705,E2 -23115.705} C_VEL
LIN {X 0,Y 170.034,Z 538.619,A -85,B 0,C 180,E1 -23118.073,E2 -23118.073} C_VEL
LIN {X 0,Y 169.506,Z 539.85,A -85,B 0,C 180,E1 -23120.453,E2 -23120.453} C_VEL
LIN {X 0,Y 169.14,Z 541.112,A -85,B 0,C 180,E1 -23125.233,E2 -23125.233} C_VEL
LIN {X 0,Y 169.238,Z 541.171,A -85,B 0,C 180,E1 -23127.619,E2 -23127.619} C_VEL
LIN {X 0,Y 169.415,Z 540.833,A -85,B 0,C 180,E1 -23129.999,E2 -23129.999} C_VEL
LIN {X 0,Y 169.306,Z 540.022,A -85,B 0,C 180,E1 -23132.378,E2 -23132.378} C_VEL
LIN {X 0,Y 169.324,Z 538.639,A -85,B 0,C 180,E1 -23135.029,E2 -23135.029} C_VEL
LIN {X 0,Y 169.63,Z 535.047,A -85,B 0,C 180,E1 -23139.539,E2 -23139.539} C_VEL
LIN {X 0,Y 170.408,Z 530.969,A -85,B 0,C 180,E1 -23143.11,E2 -23143.11} C_VEL
LIN {X 0,Y 172.127,Z 524.7,A -85,B 0,C 180,E1 -23147.218,E2 -23147.218} C_VEL
LIN {X 0,Y 174.217,Z 517.862,A -85,B 0,C 180,E1 -23150.669,E2 -23150.669} C_VEL
LIN {X 0,Y 175.945,Z 512.037,A -85,B 0,C 180,E1 -23153.053,E2 -23153.053} C_VEL
LIN {X 0,Y 176.474,Z 508.163,A -85,B 0,C 180,E1 -23154.494,E2 -23154.494} C_VEL
LIN {X 0,Y 176.085,Z 504.18,A -85,B 0,C 180,E1 -23155.93,E2 -23155.93} C_VEL
LIN {X 0,Y 173.941,Z 492.91,A -85,B 0,C 180,E1 -23159.612,E2 -23159.612} C_VEL
LIN {X 0,Y 173.861,Z 489.753,A -85,B 0,C 180,E1 -23160.465,E2 -23160.465} C_VEL
LIN {X 0,Y 173.934,Z 478.864,A -85,B 0,C 180,E1 -23163.055,E2 -23163.055} C_VEL
LIN {X 0,Y 173.392,Z 467.309,A -85,B 0,C 180,E1 -23165.374,E2 -23165.374} C_VEL
LIN {X 0,Y 172.085,Z 455.093,A -85,B 0,C 180,E1 -23167.48,E2 -23167.48} C_VEL
LIN {X 0,Y 170.005,Z 443.358,A -85,B 0,C 180,E1 -23169.258,E2 -23169.258} C_VEL
LIN {X 0,Y 168.266,Z 437.735,A -85,B 0,C 180,E1 -23170.125,E2 -23170.125} C_VEL
LIN {X 0,Y 167.005,Z 434.247,A -85,B 0,C 180,E1 -23170.662,E2 -23170.662} C_VEL
LIN {X 0,Y 166.969,Z 433.893,A -85,B 0,C 180,E1 -23170.743,E2 -23170.743} C_VEL
LIN {X 0,Y 166.207,Z 429.914,A -85,B 0,C 180,E1 -23175.957,E2 -23175.957} C_VEL
LIN {X 0,Y 165.54,Z 426.746,A -85,B 0,C 180,E1 -23180.445,E2 -23180.445} C_VEL
LIN {X 0,Y 165.128,Z 424.383,A -85,B 0,C 180,E1 -23183.962,E2 -23183.962} C_VEL
LIN {X 0,Y 164.624,Z 421.07,A -85,B 0,C 180,E1 -23189.183,E2 -23189.183} C_VEL
LIN {X 0,Y 164.387,Z 420.012,A -85,B 0,C 180,E1 -23191.251,E2 -23191.251} C_VEL
LIN {X 0,Y 164.413,Z 420.007,A -85,B 0,C 180,E1 -23194.694,E2 -23194.694} C_VEL
LIN {X 0,Y 164.482,Z 419.996,A -85,B 0,C 180,E1 -23200.049,E2 -23200.049} C_VEL
LIN {X 0,Y 164.525,Z 419.992,A -85,B 0,C 180,E1 -23205.149,E2 -23205.149} C_VEL
LIN {X 0,Y 164.763,Z 419.961,A -85,B 0,C 180,E1 -23210.176,E2 -23210.176} C_VEL
LIN {X 0,Y 164.826,Z 419.946,A -85,B 0,C 180,E1 -23212.651,E2 -23212.651} C_VEL
LIN {X 0,Y 165.043,Z 419.925,A -85,B 0,C 180,E1 -23217.56,E2 -23217.56} C_VEL
LIN {X 0,Y 165.292,Z 419.894,A -85,B 0,C 180,E1 -23220,E2 -23220} C_VEL
LIN {X 0,Y 164.825,Z 419.95,A -85,B 0,C 180,E1 -23227.102,E2 -23227.102} C_VEL
LIN {X 0,Y 164.75,Z 419.954,A -85,B 0,C 180,E1 -23231.152,E2 -23231.152} C_VEL
LIN {X 0,Y 164.481,Z 419.995,A -85,B 0,C 180,E1 -23237.404,E2 -23237.404} C_VEL
LIN {X 0,Y 164.47,Z 419.995,A -85,B 0,C 180,E1 -23239.99,E2 -23239.99} C_VEL
LIN {X 0,Y 164.39,Z 420.004,A -85,B 0,C 180,E1 -23246.135,E2 -23246.135} C_VEL
LIN {X 0,Y 164.373,Z 420,A -85,B 0,C 180,E1 -23251.229,E2 -23251.229} C_VEL
LIN {X 0,Y 164.311,Z 420.017,A -85,B 0,C 180,E1 -23256.786,E2 -23256.786} C_VEL
LIN {X 0,Y 164.3,Z 420.01,A -85,B 0,C 180,E1 -23259.914,E2 -23259.914} C_VEL
LIN {X 0,Y 164.278,Z 420.018,A -85,B 0,C 180,E1 -23263.343,E2 -23263.343} C_VEL
LIN {X 0,Y 164.291,Z 420.018,A -85,B 0,C 180,E1 -23266.81,E2 -23266.81} C_VEL
LIN {X 0,Y 164.294,Z 419.994,A -85,B 0,C 180,E1 -23270.353,E2 -23270.353} C_VEL
LIN {X 0,Y 164.329,Z 419.99,A -85,B 0,C 180,E1 -23274.35,E2 -23274.35} C_VEL
LIN {X 0,Y 164.389,Z 420.012,A -85,B 0,C 180,E1 -23279.136,E2 -23279.136} C_VEL
LIN {X 0,Y 164.417,Z 419.981,A -85,B 0,C 180,E1 -23284.695,E2 -23284.695} C_VEL
LIN {X 0,Y 164.486,Z 419.994,A -85,B 0,C 180,E1 -23290.052,E2 -23290.052} C_VEL
LIN {X 0,Y 164.556,Z 419.987,A -85,B 0,C 180,E1 -23295.153,E2 -23295.153} C_VEL
LIN {X 0,Y 164.855,Z 419.943,A -85,B 0,C 180,E1 -23300.182,E2 -23300.182} C_VEL
LIN {X 0,Y 164.852,Z 419.952,A -85,B 0,C 180,E1 -23301.342,E2 -23301.342} C_VEL
LIN {X 0,Y 165.875,Z 422.841,A -85,B 0,C 180,E1 -23301.846,E2 -23301.846} C_VEL
LIN {X 0,Y 168.402,Z 427.81,A -85,B 0,C 180,E1 -23302.933,E2 -23302.933} C_VEL
LIN {X 0,Y 171.57,Z 434.524,A -85,B 0,C 180,E1 -23304.417,E2 -23304.417} C_VEL
LIN {X 0,Y 175,Z 447.12,A -85,B 0,C 180,E1 -23307.006,E2 -23307.006} C_VEL
LIN {X 0,Y 176.645,Z 454.696,A -85,B 0,C 180,E1 -23308.705,E2 -23308.705} C_VEL
LIN {X 0,Y 177.895,Z 464.404,A -85,B 0,C 180,E1 -23311.053,E2 -23311.053} C_VEL
LIN {X 0,Y 178.086,Z 466.722,A -85,B 0,C 180,E1 -23311.657,E2 -23311.657} C_VEL
LIN {X 0,Y 175.508,Z 476.48,A -85,B 0,C 180,E1 -23313.949,E2 -23313.949} C_VEL
LIN {X 0,Y 172.929,Z 485.004,A -85,B 0,C 180,E1 -23316.417,E2 -23316.417} C_VEL
LIN {X 0,Y 170.149,Z 493.568,A -85,B 0,C 180,E1 -23319.51,E2 -23319.51} C_VEL
LIN {X 0,Y 167.506,Z 501.489,A -85,B 0,C 180,E1 -23323.164,E2 -23323.164} C_VEL
LIN {X 0,Y 165.572,Z 507.415,A -85,B 0,C 180,E1 -23326.65,E2 -23326.65} C_VEL
LIN {X 0,Y 164.1,Z 511.96,A -85,B 0,C 180,E1 -23330.037,E2 -23330.037} C_VEL
LIN {X 0,Y 163.335,Z 514.915,A -85,B 0,C 180,E1 -23332.784,E2 -23332.784} C_VEL
LIN {X 0,Y 162.648,Z 517.292,A -85,B 0,C 180,E1 -23335.601,E2 -23335.601} C_VEL
LIN {X 0,Y 162.061,Z 519.848,A -85,B 0,C 180,E1 -23339.849,E2 -23339.849} C_VEL
LIN {X 0,Y 162.167,Z 521.305,A -85,B 0,C 180,E1 -23344.57,E2 -23344.57} C_VEL
LIN {X 0,Y 162.986,Z 521.341,A -85,B 0,C 180,E1 -23349.089,E2 -23349.089} C_VEL
LIN {X 0,Y 164.448,Z 520.159,A -85,B 0,C 180,E1 -23353.403,E2 -23353.403} C_VEL
LIN {X 0,Y 166.516,Z 517.838,A -85,B 0,C 180,E1 -23357.522,E2 -23357.522} C_VEL
LIN {X 0,Y 169.539,Z 513.85,A -85,B 0,C 180,E1 -23361.963,E2 -23361.963} C_VEL
LIN {X 0,Y 173.569,Z 508.065,A -85,B 0,C 180,E1 -23366.283,E2 -23366.283} C_VEL
LIN {X 0,Y 177.148,Z 502.422,A -85,B 0,C 180,E1 -23369.411,E2 -23369.411} C_VEL
LIN {X 0,Y 181.78,Z 494.46,A -85,B 0,C 180,E1 -23372.775,E2 -23372.775} C_VEL
LIN {X 0,Y 185.902,Z 486.356,A -85,B 0,C 180,E1 -23375.427,E2 -23375.427} C_VEL
LIN {X 0,Y 188.62,Z 480.585,A -85,B 0,C 180,E1 -23376.969,E2 -23376.969} C_VEL
LIN {X 0,Y 188.863,Z 474.131,A -85,B 0,C 180,E1 -23379.296,E2 -23379.296} C_VEL
LIN {X 0,Y 188.243,Z 466.599,A -85,B 0,C 180,E1 -23382.06,E2 -23382.06} C_VEL
LIN {X 0,Y 186.796,Z 459.814,A -85,B 0,C 180,E1 -23384.73,E2 -23384.73} C_VEL
LIN {X 0,Y 184.513,Z 453.373,A -85,B 0,C 180,E1 -23387.628,E2 -23387.628} C_VEL
LIN {X 0,Y 182.344,Z 448.569,A -85,B 0,C 180,E1 -23390.088,E2 -23390.088} C_VEL
LIN {X 0,Y 180.54,Z 444.997,A -85,B 0,C 180,E1 -23392.073,E2 -23392.073} C_VEL
LIN {X 0,Y 178.086,Z 440.519,A -85,B 0,C 180,E1 -23394.906,E2 -23394.906} C_VEL
LIN {X 0,Y 175.568,Z 437.197,A -85,B 0,C 180,E1 -23397.777,E2 -23397.777} C_VEL
LIN {X 0,Y 174.691,Z 435.187,A -85,B 0,C 180,E1 -23399.159,E2 -23399.159} C_VEL
LIN {X 0,Y 171.364,Z 431.713,A -85,B 0,C 180,E1 -23403.968,E2 -23403.968} C_VEL
LIN {X 0,Y 170.912,Z 430.581,A -85,B 0,C 180,E1 -23405.042,E2 -23405.042} C_VEL
LIN {X 0,Y 168.162,Z 429.695,A -85,B 0,C 180,E1 -23412.062,E2 -23412.062} C_VEL
LIN {X 0,Y 167.823,Z 430.268,A -85,B 0,C 180,E1 -23417.046,E2 -23417.046} C_VEL
LIN {X 0,Y 168.751,Z 432.107,A -85,B 0,C 180,E1 -23422.013,E2 -23422.013} C_VEL
LIN {X 0,Y 171.135,Z 434.91,A -85,B 0,C 180,E1 -23427.087,E2 -23427.087} C_VEL
LIN {X 0,Y 172.668,Z 438.941,A -85,B 0,C 180,E1 -23430.076,E2 -23430.076} C_VEL
LIN {X 0,Y 175.199,Z 442.426,A -85,B 0,C 180,E1 -23433.262,E2 -23433.262} C_VEL
LIN {X 0,Y 176.645,Z 445.977,A -85,B 0,C 180,E1 -23435.232,E2 -23435.232} C_VEL
LIN {X 0,Y 178.317,Z 448.471,A -85,B 0,C 180,E1 -23436.946,E2 -23436.946} C_VEL
LIN {X 0,Y 179.73,Z 452.271,A -85,B 0,C 180,E1 -23438.73,E2 -23438.73} C_VEL
LIN {X 0,Y 181.181,Z 455.354,A -85,B 0,C 180,E1 -23440.253,E2 -23440.253} C_VEL
LIN {X 0,Y 184.141,Z 462.841,A -85,B 0,C 180,E1 -23443.518,E2 -23443.518} C_VEL
LIN {X 0,Y 185.588,Z 467.798,A -85,B 0,C 180,E1 -23445.369,E2 -23445.369} C_VEL
LIN {X 0,Y 186.055,Z 473.838,A -85,B 0,C 180,E1 -23447.162,E2 -23447.162} C_VEL
LIN {X 0,Y 185.763,Z 483.833,A -85,B 0,C 180,E1 -23449.972,E2 -23449.972} C_VEL
LIN {X 0,Y 184.422,Z 493.785,A -85,B 0,C 180,E1 -23452.867,E2 -23452.867} C_VEL
LIN {X 0,Y 182.488,Z 501.821,A -85,B 0,C 180,E1 -23455.385,E2 -23455.385} C_VEL
LIN {X 0,Y 180.245,Z 508.304,A -85,B 0,C 180,E1 -23457.579,E2 -23457.579} C_VEL
LIN {X 0,Y 175.737,Z 516.532,A -85,B 0,C 180,E1 -23460.666,E2 -23460.666} C_VEL
LIN {X 0,Y 171.464,Z 524.063,A -85,B 0,C 180,E1 -23464.388,E2 -23464.388} C_VEL
LIN {X 0,Y 168.267,Z 529.481,A -85,B 0,C 180,E1 -23467.92,E2 -23467.92} C_VEL
LIN {X 0,Y 165.75,Z 533.612,A -85,B 0,C 180,E1 -23471.457,E2 -23471.457} C_VEL
LIN {X 0,Y 163.855,Z 536.749,A -85,B 0,C 180,E1 -23475.087,E2 -23475.087} C_VEL
LIN {X 0,Y 163.054,Z 538.345,A -85,B 0,C 180,E1 -23477.554,E2 -23477.554} C_VEL
LIN {X 0,Y 162.168,Z 540.289,A -85,B 0,C 180,E1 -23482.529,E2 -23482.529} C_VEL
LIN {X 0,Y 162.157,Z 540.717,A -85,B 0,C 180,E1 -23487.515,E2 -23487.515} C_VEL
LIN {X 0,Y 162.351,Z 540.312,A -85,B 0,C 180,E1 -23489.999,E2 -23489.999} C_VEL
LIN {X 0,Y 162.228,Z 539.459,A -85,B 0,C 180,E1 -23492.482,E2 -23492.482} C_VEL
LIN {X 0,Y 162.254,Z 538.202,A -85,B 0,C 180,E1 -23494.969,E2 -23494.969} C_VEL
LIN {X 0,Y 162.424,Z 535.465,A -85,B 0,C 180,E1 -23498.71,E2 -23498.71} C_VEL
LIN {X 0,Y 163.116,Z 531.678,A -85,B 0,C 180,E1 -23502.44,E2 -23502.44} C_VEL
LIN {X 0,Y 164.364,Z 526.742,A -85,B 0,C 180,E1 -23506.136,E2 -23506.136} C_VEL
LIN {X 0,Y 166.322,Z 520.529,A -85,B 0,C 180,E1 -23509.757,E2 -23509.757} C_VEL
LIN {X 0,Y 168.654,Z 513.27,A -85,B 0,C 180,E1 -23513.09,E2 -23513.09} C_VEL
LIN {X 0,Y 171.394,Z 504.808,A -85,B 0,C 180,E1 -23516.154,E2 -23516.154} C_VEL
LIN {X 0,Y 173.335,Z 498.25,A -85,B 0,C 180,E1 -23518.12,E2 -23518.12} C_VEL
LIN {X 0,Y 173.861,Z 489.753,A -85,B 0,C 180,E1 -23520.465,E2 -23520.465} C_VEL
LIN {X 0,Y 173.351,Z 485.221,A -85,B 0,C 180,E1 -23521.702,E2 -23521.702} C_VEL
LIN {X 0,Y 170.626,Z 477.996,A -85,B 0,C 180,E1 -23523.777,E2 -23523.777} C_VEL
LIN {X 0,Y 167.633,Z 470.501,A -85,B 0,C 180,E1 -23525.776,E2 -23525.776} C_VEL
LIN {X 0,Y 166.684,Z 465.53,A -85,B 0,C 180,E1 -23526.856,E2 -23526.856} C_VEL
LIN {X 0,Y 165.401,Z 454.064,A -85,B 0,C 180,E1 -23528.912,E2 -23528.912} C_VEL
LIN {X 0,Y 163.581,Z 444.243,A -85,B 0,C 180,E1 -23530.501,E2 -23530.501} C_VEL
LIN {X 0,Y 161.094,Z 437.391,A -85,B 0,C 180,E1 -23531.731,E2 -23531.731} C_VEL
LIN {X 0,Y 159.913,Z 434.647,A -85,B 0,C 180,E1 -23532.247,E2 -23532.247} C_VEL
LIN {X 0,Y 159.681,Z 433.385,A -85,B 0,C 180,E1 -23532.448,E2 -23532.448} C_VEL
LIN {X 0,Y 159.036,Z 430.317,A -85,B 0,C 180,E1 -23536.767,E2 -23536.767} C_VEL
LIN {X 0,Y 158.214,Z 426.093,A -85,B 0,C 180,E1 -23543.087,E2 -23543.087} C_VEL
LIN {X 0,Y 157.712,Z 423.165,A -85,B 0,C 180,E1 -23547.849,E2 -23547.849} C_VEL
LIN {X 0,Y 157.317,Z 420.893,A -85,B 0,C 180,E1 -23552.027,E2 -23552.027} C_VEL
LIN {X 0,Y 157.311,Z 420.89,A -85,B 0,C 180,E1 -23556.292,E2 -23556.292} C_VEL
LIN {X 0,Y 157.415,Z 420.876,A -85,B 0,C 180,E1 -23561.789,E2 -23561.789} C_VEL
LIN {X 0,Y 157.527,Z 420.863,A -85,B 0,C 180,E1 -23567.111,E2 -23567.111} C_VEL
LIN {X 0,Y 157.685,Z 420.842,A -85,B 0,C 180,E1 -23569.731,E2 -23569.731} C_VEL
LIN {X 0,Y 157.763,Z 420.828,A -85,B 0,C 180,E1 -23572.32,E2 -23572.32} C_VEL
LIN {X 0,Y 158.254,Z 420.771,A -85,B 0,C 180,E1 -23580,E2 -23580} C_VEL
LIN {X 0,Y 157.807,Z 420.827,A -85,B 0,C 180,E1 -23587.678,E2 -23587.678} C_VEL
LIN {X 0,Y 157.679,Z 420.835,A -85,B 0,C 180,E1 -23591.32,E2 -23591.32} C_VEL
LIN {X 0,Y 157.457,Z 420.866,A -85,B 0,C 180,E1 -23595.534,E2 -23595.534} C_VEL
LIN {X 0,Y 157.367,Z 420.874,A -85,B 0,C 180,E1 -23600.934,E2 -23600.934} C_VEL
LIN {X 0,Y 157.312,Z 420.889,A -85,B 0,C 180,E1 -23606.686,E2 -23606.686} C_VEL
LIN {X 0,Y 157.276,Z 420.879,A -85,B 0,C 180,E1 -23612.428,E2 -23612.428} C_VEL
LIN {X 0,Y 157.281,Z 420.894,A -85,B 0,C 180,E1 -23616.458,E2 -23616.458} C_VEL
LIN {X 0,Y 157.212,Z 420.891,A -85,B 0,C 180,E1 -23622.111,E2 -23622.111} C_VEL
LIN {X 0,Y 157.21,Z 420.895,A -85,B 0,C 180,E1 -23627.891,E2 -23627.891} C_VEL
LIN {X 0,Y 157.267,Z 420.86,A -85,B 0,C 180,E1 -23633.552,E2 -23633.552} C_VEL
LIN {X 0,Y 157.292,Z 420.896,A -85,B 0,C 180,E1 -23638.098,E2 -23638.098} C_VEL
LIN {X 0,Y 157.322,Z 420.866,A -85,B 0,C 180,E1 -23643.467,E2 -23643.467} C_VEL
LIN {X 0,Y 157.396,Z 420.879,A -85,B 0,C 180,E1 -23649.668,E2 -23649.668} C_VEL
LIN {X 0,Y 157.48,Z 420.86,A -85,B 0,C 180,E1 -23654.47,E2 -23654.47} C_VEL
LIN {X 0,Y 157.798,Z 420.99,A -85,B 0,C 180,E1 -23659.739,E2 -23659.739} C_VEL
LIN {X 0,Y 158.925,Z 423.807,A -85,B 0,C 180,E1 -23660.29,E2 -23660.29} C_VEL
LIN {X 0,Y 163.029,Z 431.99,A -85,B 0,C 180,E1 -23662.227,E2 -23662.227} C_VEL
LIN {X 0,Y 166.367,Z 439.875,A -85,B 0,C 180,E1 -23664.082,E2 -23664.082} C_VEL
LIN {X 0,Y 169.319,Z 451.891,A -85,B 0,C 180,E1 -23666.81,E2 -23666.81} C_VEL
LIN {X 0,Y 170.878,Z 461.478,A -85,B 0,C 180,E1 -23669.17,E2 -23669.17} C_VEL
LIN {X 0,Y 171.469,Z 467.949,A -85,B 0,C 180,E1 -23670.881,E2 -23670.881} C_VEL
LIN {X 0,Y 168.673,Z 477.826,A -85,B 0,C 180,E1 -23673.317,E2 -23673.317} C_VEL
LIN {X 0,Y 165.808,Z 486.772,A -85,B 0,C 180,E1 -23676.083,E2 -23676.083} C_VEL
LIN {X 0,Y 163.05,Z 494.814,A -85,B 0,C 180,E1 -23679.189,E2 -23679.189} C_VEL
LIN {X 0,Y 160.572,Z 501.934,A -85,B 0,C 180,E1 -23682.641,E2 -23682.641} C_VEL
LIN {X 0,Y 158.345,Z 508.576,A -85,B 0,C 180,E1 -23686.768,E2 -23686.768} C_VEL
LIN {X 0,Y 156.709,Z 513.719,A -85,B 0,C 180,E1 -23691.025,E2 -23691.025} C_VEL
LIN {X 0,Y 155.579,Z 517.553,A -85,B 0,C 180,E1 -23695.381,E2 -23695.381} C_VEL
LIN {X 0,Y 154.963,Z 520.486,A -85,B 0,C 180,E1 -23700.491,E2 -23700.491} C_VEL
LIN {X 0,Y 155.153,Z 521.789,A -85,B 0,C 180,E1 -23705.377,E2 -23705.377} C_VEL
LIN {X 0,Y 156.139,Z 521.742,A -85,B 0,C 180,E1 -23710.075,E2 -23710.075} C_VEL
LIN {X 0,Y 158.153,Z 520.168,A -85,B 0,C 180,E1 -23715.317,E2 -23715.317} C_VEL
LIN {X 0,Y 160.849,Z 517.192,A -85,B 0,C 180,E1 -23720.012,E2 -23720.012} C_VEL
LIN {X 0,Y 164.297,Z 512.913,A -85,B 0,C 180,E1 -23724.364,E2 -23724.364} C_VEL
LIN {X 0,Y 167.906,Z 507.977,A -85,B 0,C 180,E1 -23727.951,E2 -23727.951} C_VEL
LIN {X 0,Y 172.24,Z 501.49,A -85,B 0,C 180,E1 -23731.468,E2 -23731.468} C_VEL
LIN {X 0,Y 177.202,Z 493.196,A -85,B 0,C 180,E1 -23734.87,E2 -23734.87} C_VEL
LIN {X 0,Y 181.411,Z 485.347,A -85,B 0,C 180,E1 -23737.354,E2 -23737.354} C_VEL
LIN {X 0,Y 182.819,Z 482.424,A -85,B 0,C 180,E1 -23738.154,E2 -23738.154} C_VEL
LIN {X 0,Y 183.177,Z 475.18,A -85,B 0,C 180,E1 -23740.966,E2 -23740.966} C_VEL
LIN {X 0,Y 182.595,Z 468.208,A -85,B 0,C 180,E1 -23743.796,E2 -23743.796} C_VEL
LIN {X 0,Y 181.219,Z 462,A -85,B 0,C 180,E1 -23746.544,E2 -23746.544} C_VEL
LIN {X 0,Y 178.908,Z 455.528,A -85,B 0,C 180,E1 -23749.896,E2 -23749.896} C_VEL
LIN {X 0,Y 176.505,Z 450.111,A -85,B 0,C 180,E1 -23753.139,E2 -23753.139} C_VEL
LIN {X 0,Y 174.852,Z 446.748,A -85,B 0,C 180,E1 -23755.389,E2 -23755.389} C_VEL
LIN {X 0,Y 173.088,Z 444.319,A -85,B 0,C 180,E1 -23757.673,E2 -23757.673} C_VEL
LIN {X 0,Y 171.717,Z 441.405,A -85,B 0,C 180,E1 -23760,E2 -23760} C_VEL
LIN {X 0,Y 168.991,Z 438,A -85,B 0,C 180,E1 -23764.771,E2 -23764.771} C_VEL
LIN {X 0,Y 168.775,Z 437.364,A -85,B 0,C 180,E1 -23765.436,E2 -23765.436} C_VEL
LIN {X 0,Y 166.423,Z 436.564,A -85,B 0,C 180,E1 -23772.189,E2 -23772.189} C_VEL
LIN {X 0,Y 166.128,Z 437.23,A -85,B 0,C 180,E1 -23777.225,E2 -23777.225} C_VEL
LIN {X 0,Y 167.188,Z 439.324,A -85,B 0,C 180,E1 -23782.635,E2 -23782.635} C_VEL
LIN {X 0,Y 168.824,Z 441.417,A -85,B 0,C 180,E1 -23786.417,E2 -23786.417} C_VEL
LIN {X 0,Y 170.432,Z 445.888,A -85,B 0,C 180,E1 -23790.008,E2 -23790.008} C_VEL
LIN {X 0,Y 172.196,Z 448.585,A -85,B 0,C 180,E1 -23792.536,E2 -23792.536} C_VEL
LIN {X 0,Y 173.433,Z 451.969,A -85,B 0,C 180,E1 -23794.563,E2 -23794.563} C_VEL
LIN {X 0,Y 174.431,Z 453.61,A -85,B 0,C 180,E1 -23795.749,E2 -23795.749} C_VEL
LIN {X 0,Y 177.523,Z 461.857,A -85,B 0,C 180,E1 -23800.041,E2 -23800.041} C_VEL
LIN {X 0,Y 179.872,Z 468.764,A -85,B 0,C 180,E1 -23803.212,E2 -23803.212} C_VEL
LIN {X 0,Y 180.734,Z 472.934,A -85,B 0,C 180,E1 -23804.814,E2 -23804.814} C_VEL
LIN {X 0,Y 180.557,Z 481.406,A -85,B 0,C 180,E1 -23807.394,E2 -23807.394} C_VEL
LIN {X 0,Y 179.317,Z 491.478,A -85,B 0,C 180,E1 -23810.481,E2 -23810.481} C_VEL
LIN {X 0,Y 177.501,Z 499.527,A -85,B 0,C 180,E1 -23813.068,E2 -23813.068} C_VEL
LIN {X 0,Y 174.905,Z 507.235,A -85,B 0,C 180,E1 -23815.768,E2 -23815.768} C_VEL
LIN {X 0,Y 171.887,Z 512.929,A -85,B 0,C 180,E1 -23817.891,E2 -23817.891} C_VEL
LIN {X 0,Y 167.475,Z 520.221,A -85,B 0,C 180,E1 -23821.145,E2 -23821.145} C_VEL
LIN {X 0,Y 163.892,Z 526.148,A -85,B 0,C 180,E1 -23824.607,E2 -23824.607} C_VEL
LIN {X 0,Y 160.732,Z 530.896,A -85,B 0,C 180,E1 -23828.182,E2 -23828.182} C_VEL
LIN {X 0,Y 158.247,Z 534.589,A -85,B 0,C 180,E1 -23831.887,E2 -23831.887} C_VEL
LIN {X 0,Y 156.959,Z 536.536,A -85,B 0,C 180,E1 -23834.415,E2 -23834.415} C_VEL
LIN {X 0,Y 155.455,Z 539.166,A -85,B 0,C 180,E1 -23839.581,E2 -23839.581} C_VEL
LIN {X 0,Y 154.992,Z 540.276,A -85,B 0,C 180,E1 -23844.796,E2 -23844.796} C_VEL
LIN {X 0,Y 155.079,Z 540.24,A -85,B 0,C 180,E1 -23847.402,E2 -23847.402} C_VEL
LIN {X 0,Y 155.286,Z 539.779,A -85,B 0,C 180,E1 -23849.999,E2 -23849.999} C_VEL
LIN {X 0,Y 155.176,Z 537.766,A -85,B 0,C 180,E1 -23854.869,E2 -23854.869} C_VEL
LIN {X 0,Y 155.41,Z 534.767,A -85,B 0,C 180,E1 -23859.106,E2 -23859.106} C_VEL
LIN {X 0,Y 156.166,Z 530.889,A -85,B 0,C 180,E1 -23863.003,E2 -23863.003} C_VEL
LIN {X 0,Y 157.537,Z 525.859,A -85,B 0,C 180,E1 -23866.855,E2 -23866.855} C_VEL
LIN {X 0,Y 159.59,Z 519.523,A -85,B 0,C 180,E1 -23870.627,E2 -23870.627} C_VEL
LIN {X 0,Y 161.834,Z 512.92,A -85,B 0,C 180,E1 -23873.745,E2 -23873.745} C_VEL
LIN {X 0,Y 164.427,Z 505.265,A -85,B 0,C 180,E1 -23876.665,E2 -23876.665} C_VEL
LIN {X 0,Y 166.457,Z 498.801,A -85,B 0,C 180,E1 -23878.701,E2 -23878.701} C_VEL
LIN {X 0,Y 167.142,Z 488.766,A -85,B 0,C 180,E1 -23881.615,E2 -23881.615} C_VEL
LIN {X 0,Y 167.263,Z 478.323,A -85,B 0,C 180,E1 -23884.192,E2 -23884.192} C_VEL
LIN {X 0,Y 166.87,Z 467.716,A -85,B 0,C 180,E1 -23886.433,E2 -23886.433} C_VEL
LIN {X 0,Y 166.684,Z 465.53,A -85,B 0,C 180,E1 -23886.856,E2 -23886.856} C_VEL
LIN {X 0,Y 165.739,Z 460.511,A -85,B 0,C 180,E1 -23887.891,E2 -23887.891} C_VEL
LIN {X 0,Y 163.914,Z 455.794,A -85,B 0,C 180,E1 -23888.981,E2 -23888.981} C_VEL
